C05453=1098.918,347.540,412.649,179.010,19.084,152.317
C05454=1098.913,347.292,412.684,179.007,19.081,152.317
C05455=1098.907,347.044,412.717,179.003,19.078,152.317
C05456=1098.902,346.797,412.751,179.000,19.074,152.316
C05457=1098.895,346.549,412.786,178.998,19.071,152.316
C05458=1098.890,346.301,412.819,178.994,19.067,152.316
C05459=1098.884,346.054,412.853,178.992,19.064,152.316
C05460=1098.879,345.806,412.888,178.988,19.060,152.315
C05461=1098.873,345.558,412.921,178.985,19.057,152.315
C05462=1098.867,345.311,412.955,178.982,19.053,152.315
C05463=1098.862,345.063,412.989,178.979,19.050,152.314
C05464=1098.856,344.816,413.023,178.976,19.046,152.314
C05465=1098.850,344.568,413.056,178.973,19.043,152.314
C05466=1098.844,344.320,413.090,178.969,19.039,152.314
C05467=1098.839,344.073,413.123,178.966,19.036,152.313
C05468=1098.829,343.698,413.175,178.962,19.031,152.313
C05469=1098.821,343.324,413.226,178.957,19.026,152.313
C05470=1098.812,342.950,413.276,178.952,19.021,152.312
C05471=1098.804,342.576,413.327,178.947,19.015,152.312
C05472=1098.798,342.328,413.360,178.945,19.012,152.312
C05473=1098.793,342.080,413.394,178.941,19.008,152.311
C05474=1098.787,341.833,413.428,178.938,19.006,152.311
C05475=1098.781,341.585,413.461,178.935,19.003,152.311
C05476=1098.776,341.337,413.495,178.932,18.999,152.311
C05477=1098.770,341.089,413.528,178.929,18.996,152.311
C05478=1098.764,340.842,413.562,178.925,18.992,152.310
C05479=1098.759,340.594,413.596,178.923,18.989,152.310
C05480=1098.753,340.346,413.629,178.920,18.986,152.310
C05481=1098.747,340.099,413.662,178.916,18.982,152.310
C05482=1098.741,339.851,413.695,178.913,18.979,152.310
C05483=1098.736,339.603,413.729,178.910,18.975,152.309
C05484=1098.730,339.356,413.763,178.907,18.972,152.309
C05485=1098.724,339.108,413.796,178.904,18.970,152.309
C05486=1098.719,338.860,413.829,178.901,18.966,152.309
C05487=1098.713,338.612,413.863,178.898,18.963,152.308
C05488=1098.707,338.364,413.895,178.895,18.960,152.308
C05489=1098.701,338.116,413.929,178.891,18.956,152.308
C05490=1098.696,337.869,413.962,178.888,18.953,152.308
C05491=1098.690,337.621,413.996,178.885,18.950,152.308
C05492=1098.684,337.374,414.029,178.882,18.947,152.308
C05493=1098.678,337.126,414.062,178.879,18.944,152.307
C05494=1098.672,336.878,414.096,178.875,18.940,152.307
C05495=1098.667,336.630,414.129,178.872,18.937,152.307
C05496=1098.661,336.382,414.162,178.870,18.934,152.307
C05497=1098.656,336.135,414.195,178.866,18.931,152.307
C05498=1098.650,335.887,414.228,178.863,18.928,152.306
C05499=1098.644,335.640,414.261,178.860,18.925,152.306
C05500=1098.638,335.392,414.294,178.856,18.921,152.306
C05501=1098.633,335.144,414.327,178.853,18.919,152.306
C05502=1098.627,334.896,414.359,178.851,18.915,152.306
C05503=1098.621,334.648,414.393,178.848,18.913,152.306
C05504=1098.616,334.400,414.426,178.844,18.909,152.305
C05505=1098.610,334.153,414.458,178.841,18.906,152.305
C05506=1098.604,333.905,414.492,178.838,18.903,152.305
C05507=1098.599,333.657,414.525,178.834,18.900,152.305
C05508=1098.593,333.410,414.558,178.831,18.897,152.305
C05509=1098.587,333.161,414.590,178.829,18.894,152.305
C05510=1098.582,332.913,414.624,178.825,18.891,152.305
C05511=1098.576,332.666,414.656,178.822,18.888,152.304
C05512=1098.570,332.418,414.689,178.819,18.885,152.304
C05513=1098.564,332.170,414.722,178.815,18.881,152.304
C05514=1098.559,331.922,414.755,178.812,18.879,152.304
C05515=1098.553,331.675,414.788,178.809,18.876,152.304
C05516=1098.547,331.427,414.821,178.806,18.873,152.304
C05517=1098.542,331.179,414.853,178.803,18.870,152.304
C05518=1098.535,330.932,414.885,178.800,18.867,152.304
C05519=1098.530,330.684,414.919,178.797,18.864,152.303
C05520=1098.520,330.303,414.969,178.791,18.859,152.303
C05521=1098.511,329.923,415.019,178.787,18.855,152.303
C05522=1098.504,329.542,415.068,178.781,18.851,152.303
C05523=1098.494,329.162,415.119,178.777,18.846,152.303
C05524=1098.488,328.915,415.151,178.774,18.844,152.303
C05525=1098.483,328.666,415.184,178.770,18.840,152.303
C05526=1098.477,328.419,415.216,178.767,18.838,152.303
C05527=1098.471,328.170,415.248,178.764,18.835,152.303
C05528=1098.465,327.923,415.281,178.761,18.832,152.302
C05529=1098.460,327.675,415.313,178.757,18.829,152.302
C05530=1098.454,327.427,415.346,178.754,18.826,152.302
C05531=1098.448,327.179,415.378,178.751,18.823,152.302
C05532=1098.442,326.931,415.411,178.748,18.821,152.302
C05533=1098.437,326.684,415.443,178.745,18.818,152.302
C05534=1098.430,326.436,415.476,178.742,18.815,152.302
C05535=1098.424,326.188,415.508,178.738,18.812,152.302
C05536=1098.420,325.940,415.540,178.735,18.810,152.302
C05537=1098.413,325.693,415.573,178.732,18.807,152.302
C05538=1098.407,325.444,415.605,178.729,18.803,152.302
C05539=1098.402,325.197,415.637,178.726,18.801,152.302
C05540=1098.397,324.949,415.670,178.723,18.798,152.301
C05541=1098.391,324.701,415.702,178.720,18.795,152.301
C05542=1098.385,324.453,415.734,178.717,18.793,152.301
C05543=1098.379,324.206,415.766,178.713,18.790,152.301
C05544=1098.374,323.957,415.799,178.710,18.787,152.301
C05545=1098.368,323.710,415.831,178.707,18.784,152.301
C05546=1098.362,323.461,415.863,178.704,18.781,152.301
C05547=1098.356,323.214,415.895,178.701,18.779,152.301
C05548=1098.351,322.966,415.927,178.698,18.776,152.301
C05549=1098.345,322.718,415.960,178.693,18.773,152.301
C05550=1098.340,322.470,415.991,178.690,18.770,152.301
C05551=1098.334,322.222,416.023,178.687,18.768,152.301
C05552=1098.329,322.012,416.050,178.684,18.765,152.301
C05553=1098.324,321.802,416.078,178.682,18.763,152.301
C05554=1098.320,321.592,416.105,178.679,18.760,152.301
C05555=1098.315,321.381,416.132,178.677,18.759,152.301
C05556=1098.310,321.171,416.159,178.674,18.756,152.301
C05557=1098.306,320.961,416.186,178.671,18.754,152.300
C05558=1098.301,320.751,416.213,178.668,18.752,152.301
C05559=1098.296,320.541,416.240,178.666,18.749,152.300
C05560=1098.290,320.293,416.272,178.663,18.747,152.300
C05561=1098.285,320.045,416.304,178.659,18.744,152.300
C05562=1098.279,319.797,416.336,178.656,18.741,152.300
C05563=1098.273,319.549,416.368,178.653,18.738,152.300
C05564=1098.267,319.301,416.400,178.650,18.736,152.300
C05565=1098.262,319.054,416.432,178.647,18.733,152.300
C05566=1098.256,318.805,416.464,178.644,18.731,152.300
C05567=1098.251,318.558,416.495,178.640,18.728,152.300
C05568=1098.245,318.310,416.527,178.637,18.725,152.300
C05569=1098.239,318.062,416.559,178.634,18.722,152.300
C05570=1098.234,317.814,416.592,178.630,18.720,152.300
C05571=1098.229,317.566,416.623,178.627,18.717,152.300
C05572=1098.223,317.334,416.652,178.624,18.715,152.300
C05573=1098.218,317.104,416.682,178.621,18.712,152.300
C05574=1098.213,316.872,416.712,178.618,18.709,152.300
C05575=1098.207,316.640,416.741,178.616,18.708,152.300
C05576=1098.203,316.409,416.771,178.613,18.705,152.300
C05577=1098.198,316.177,416.800,178.609,18.703,152.300
C05578=1098.191,315.946,416.830,178.606,18.700,152.300
C05579=1098.187,315.715,416.859,178.603,18.698,152.300
C05580=1098.181,315.467,416.891,178.600,18.695,152.300
C05581=1098.176,315.219,416.923,178.597,18.692,152.300
C05582=1098.170,314.971,416.955,178.594,18.690,152.300
C05583=1098.164,314.723,416.986,178.591,18.687,152.300
C05584=1098.158,314.475,417.017,178.587,18.685,152.300
C05585=1098.152,314.227,417.049,178.584,18.682,152.300
C05586=1098.147,313.979,417.080,178.581,18.680,152.300
C05587=1098.141,313.731,417.111,178.578,18.678,152.300
C05588=1098.135,313.484,417.143,178.574,18.675,152.300
C05589=1098.129,313.235,417.174,178.571,18.673,152.300
C05590=1098.123,312.988,417.205,178.568,18.670,152.300
C05591=1098.117,312.740,417.237,178.564,18.668,152.300
C05592=1098.112,312.492,417.268,178.561,18.665,152.300
C05593=1098.106,312.244,417.300,178.558,18.663,152.300
C05594=1098.100,311.995,417.331,178.555,18.661,152.300
C05595=1098.095,311.748,417.362,178.552,18.658,152.300
C05596=1098.089,311.499,417.393,178.548,18.656,152.300
C05597=1098.083,311.252,417.425,178.545,18.653,152.300
C05598=1098.077,311.004,417.456,178.542,18.651,152.300
C05599=1098.072,310.756,417.487,178.539,18.649,152.300
C05600=1098.066,310.508,417.519,178.535,18.646,152.300
C05601=1098.060,310.260,417.549,178.532,18.644,152.300
C05602=1098.055,310.012,417.580,178.528,18.641,152.300
C05603=1098.048,309.765,417.611,178.525,18.639,152.300
C05604=1098.043,309.516,417.643,178.522,18.636,152.300
C05605=1098.037,309.268,417.674,178.519,18.634,152.301
C05606=1098.032,309.020,417.705,178.515,18.632,152.301
C05607=1098.026,308.773,417.736,178.512,18.629,152.301
C05608=1098.020,308.524,417.767,178.509,18.627,152.301
C05609=1098.015,308.276,417.798,178.506,18.624,152.301
C05610=1098.009,308.029,417.829,178.503,18.622,152.301
C05611=1098.003,307.780,417.860,178.499,18.620,152.301
C05612=1097.997,307.532,417.891,178.496,18.617,152.301
C05613=1097.992,307.285,417.922,178.493,18.615,152.301
C05614=1097.986,307.037,417.953,178.490,18.613,152.301
C05615=1097.980,306.788,417.984,178.486,18.610,152.301
C05616=1097.974,306.540,418.014,178.483,18.608,152.301
C05617=1097.969,306.293,418.046,178.480,18.606,152.301
C05618=1097.963,306.045,418.076,178.477,18.604,152.301
C05619=1097.958,305.797,418.107,178.473,18.601,152.301
C05620=1097.952,305.548,418.138,178.470,18.599,152.301
C05621=1097.946,305.301,418.170,178.467,18.597,152.301
C05622=1097.941,305.053,418.200,178.464,18.594,152.301
C05623=1097.935,304.805,418.231,178.460,18.592,152.302
C05624=1097.930,304.557,418.261,178.457,18.590,152.302
C05625=1097.924,304.308,418.293,178.453,18.587,152.302
C05626=1097.918,304.060,418.323,178.450,18.585,152.302
C05627=1097.912,303.813,418.353,178.447,18.582,152.302
C05628=1097.904,303.428,418.402,178.442,18.579,152.302
C05629=1097.895,303.043,418.449,178.437,18.575,152.302
C05630=1097.887,302.658,418.497,178.432,18.572,152.302
C05631=1097.878,302.274,418.545,178.427,18.568,152.302
C05632=1097.872,302.026,418.575,178.424,18.566,152.302
C05633=1097.867,301.778,418.606,178.421,18.564,152.302
C05634=1097.861,301.530,418.636,178.417,18.562,152.302
C05635=1097.855,301.282,418.666,178.414,18.559,152.302
C05636=1097.850,301.034,418.697,178.411,18.557,152.303
C05637=1097.845,300.786,418.727,178.408,18.555,152.303
C05638=1097.839,300.538,418.758,178.404,18.552,152.303
C05639=1097.834,300.290,418.789,178.401,18.550,152.303
C05640=1097.827,300.041,418.819,178.398,18.548,152.303
C05641=1097.821,299.793,418.850,178.395,18.545,152.303
C05642=1097.816,299.545,418.881,178.391,18.543,152.303
C05643=1097.811,299.298,418.911,178.388,18.541,152.303
C05644=1097.805,299.049,418.941,178.385,18.539,152.303
C05645=1097.800,298.801,418.972,178.381,18.537,152.303
C05646=1097.794,298.553,419.002,178.378,18.534,152.303
C05647=1097.788,298.305,419.032,178.375,18.532,152.303
C05648=1097.782,298.057,419.063,178.372,18.530,152.303
C05649=1097.778,297.809,419.093,178.368,18.527,152.304
C05650=1097.772,297.561,419.123,178.365,18.526,152.304
C05651=1097.766,297.313,419.154,178.362,18.523,152.304
C05652=1097.761,297.065,419.183,178.358,18.521,152.304
C05653=1097.755,296.817,419.213,178.355,18.519,152.304
C05654=1097.749,296.569,419.244,178.352,18.517,152.304
C05655=1097.743,296.321,419.274,178.348,18.515,152.304
C05656=1097.738,296.073,419.304,178.345,18.512,152.304
C05657=1097.732,295.825,419.334,178.342,18.510,152.305
C05658=1097.727,295.576,419.364,178.338,18.508,152.305
C05659=1097.721,295.328,419.395,178.335,18.506,152.305
C05660=1097.715,295.081,419.425,178.332,18.504,152.305
C05661=1097.710,294.832,419.455,178.328,18.502,152.305
C05662=1097.704,294.584,419.485,178.325,18.499,152.305
C05663=1097.699,294.336,419.515,178.322,18.498,152.305
C05664=1097.693,294.088,419.545,178.319,18.496,152.305
C05665=1097.687,293.840,419.575,178.316,18.494,152.306
C05666=1097.681,293.592,419.605,178.312,18.492,152.306
C05667=1097.676,293.344,419.635,178.309,18.489,152.306
C05668=1097.670,293.095,419.665,178.306,18.487,152.306
C05669=1097.665,292.847,419.695,178.302,18.485,152.306
C05670=1097.659,292.599,419.725,178.299,18.483,152.306
C05671=1097.652,292.351,419.754,178.296,18.481,152.306
C05672=1097.647,292.103,419.784,178.292,18.479,152.306
C05673=1097.641,291.855,419.814,178.289,18.477,152.307
C05674=1097.635,291.607,419.844,178.286,18.474,152.307
C05675=1097.630,291.359,419.874,178.283,18.473,152.307
C05676=1097.625,291.111,419.903,178.280,18.471,152.307
C05677=1097.619,290.863,419.934,178.276,18.469,152.307
C05678=1097.614,290.615,419.963,178.273,18.467,152.307
C05679=1097.608,290.366,419.993,178.269,18.465,152.307
C05680=1097.600,289.996,420.037,178.264,18.461,152.308
C05681=1097.590,289.625,420.082,178.259,18.458,152.308
C05682=1097.582,289.254,420.126,178.255,18.456,152.308
C05683=1097.574,288.883,420.171,178.250,18.453,152.308
C05684=1097.568,288.635,420.200,178.247,18.451,152.308
C05685=1097.562,288.386,420.229,178.243,18.449,152.309
C05686=1097.557,288.139,420.260,178.240,18.447,152.309
C05687=1097.551,287.890,420.289,178.236,18.445,152.309
C05688=1097.545,287.642,420.318,178.233,18.443,152.309
C05689=1097.539,287.394,420.348,178.230,18.441,152.309
C05690=1097.534,287.145,420.378,178.227,18.439,152.309
C05691=1097.528,286.898,420.406,178.224,18.437,152.310
C05692=1097.522,286.650,420.437,178.220,18.435,152.310
C05693=1097.517,286.402,420.466,178.217,18.433,152.310
C05694=1097.511,286.153,420.496,178.213,18.431,152.310
C05695=1097.505,285.905,420.525,178.210,18.429,152.310
C05696=1097.500,285.657,420.555,178.207,18.427,152.310
C05697=1097.495,285.409,420.584,178.204,18.425,152.311
C05698=1097.488,285.161,420.613,178.200,18.424,152.311
C05699=1097.483,284.912,420.643,178.197,18.421,152.311
C05700=1097.477,284.664,420.672,178.194,18.419,152.311
C05701=1097.471,284.416,420.701,178.190,18.418,152.311
C05702=1097.466,284.168,420.731,178.187,18.415,152.311
C05703=1097.461,283.919,420.760,178.183,18.413,152.312
C05704=1097.455,283.671,420.789,178.181,18.412,152.312
C05705=1097.449,283.423,420.819,178.177,18.410,152.312
C05706=1097.443,283.175,420.848,178.174,18.408,152.312
C05707=1097.438,282.927,420.877,178.171,18.406,152.312
C05708=1097.432,282.679,420.907,178.167,18.404,152.312
C05709=1097.426,282.430,420.935,178.164,18.402,152.313
C05710=1097.422,282.182,420.964,178.161,18.400,152.313
C05711=1097.415,281.934,420.993,178.158,18.398,152.313
C05712=1097.410,281.685,421.023,178.154,18.397,152.313
C05713=1097.405,281.438,421.052,178.151,18.394,152.313
C05714=1097.399,281.190,421.081,178.147,18.392,152.313
C05715=1097.393,280.941,421.110,178.144,18.391,152.314
C05716=1097.387,280.692,421.139,178.142,18.389,152.314
C05717=1097.382,280.445,421.169,178.138,18.387,152.314
C05718=1097.376,280.197,421.198,178.134,18.385,152.314
C05719=1097.370,279.948,421.226,178.131,18.383,152.314
C05720=1097.365,279.699,421.256,178.127,18.381,152.315
C05721=1097.359,279.452,421.284,178.125,18.380,152.315
C05722=1097.353,279.203,421.314,178.122,18.378,152.315
C05723=1097.347,278.955,421.342,178.118,18.376,152.315
C05724=1097.343,278.707,421.372,178.115,18.374,152.315
C05725=1097.336,278.459,421.401,178.111,18.372,152.316
C05726=1097.330,278.210,421.429,178.109,18.371,152.316
C05727=1097.325,277.962,421.458,178.105,18.369,152.316
C05728=1097.319,277.714,421.487,178.102,18.367,152.316
C05729=1097.314,277.465,421.516,178.098,18.365,152.316
C05730=1097.308,277.218,421.545,178.095,18.363,152.316
C05731=1097.302,276.969,421.573,178.092,18.361,152.317
C05732=1097.294,276.607,421.615,178.087,18.359,152.317
C05733=1097.286,276.247,421.657,178.082,18.356,152.317
C05734=1097.278,275.884,421.699,178.077,18.353,152.318
C05735=1097.270,275.523,421.741,178.072,18.350,152.318
C05736=1097.264,275.274,421.770,178.069,18.349,152.318
C05737=1097.258,275.026,421.799,178.066,18.347,152.318
C05738=1097.253,274.778,421.827,178.062,18.345,152.319
C05739=1097.247,274.530,421.856,178.059,18.344,152.319
C05740=1097.242,274.282,421.884,178.056,18.342,152.319
C05741=1097.236,274.034,421.913,178.053,18.340,152.319
C05742=1097.230,273.786,421.941,178.049,18.338,152.319
C05743=1097.224,273.537,421.970,178.046,18.336,152.320
C05744=1097.219,273.288,421.999,178.042,18.334,152.320
C05745=1097.214,273.040,422.027,178.040,18.333,152.320
C05746=1097.208,272.792,422.056,178.036,18.331,152.320
C05747=1097.202,272.544,422.084,178.033,18.330,152.321
C05748=1097.196,272.295,422.113,178.029,18.328,152.321
C05749=1097.190,272.047,422.141,178.026,18.326,152.321
C05750=1097.185,271.799,422.170,178.023,18.325,152.321
C05751=1097.179,271.550,422.199,178.019,18.323,152.321
C05752=1097.174,271.302,422.226,178.016,18.321,152.322
C05753=1097.168,271.053,422.255,178.014,18.319,152.322
C05754=1097.162,270.806,422.283,178.010,18.317,152.322
C05755=1097.156,270.557,422.312,178.006,18.315,152.322
C05756=1097.151,270.309,422.340,178.003,18.314,152.322
C05757=1097.145,270.060,422.368,178.000,18.312,152.323
C05758=1097.140,269.813,422.397,177.997,18.310,152.323
C05759=1097.134,269.564,422.426,177.993,18.309,152.323
C05760=1097.129,269.316,422.454,177.990,18.307,152.323
C05761=1097.123,269.067,422.482,177.987,18.305,152.324
C05762=1097.118,268.819,422.510,177.984,18.304,152.324
C05763=1097.112,268.570,422.538,177.980,18.302,152.324
C05764=1097.106,268.322,422.566,177.977,18.300,152.324
C05765=1097.100,268.073,422.595,177.974,18.299,152.324
C05766=1097.095,267.825,422.622,177.970,18.297,152.325
C05767=1097.089,267.577,422.652,177.967,18.295,152.325
C05768=1097.083,267.329,422.679,177.964,18.294,152.325
C05769=1097.078,267.080,422.708,177.961,18.292,152.325
C05770=1097.072,266.832,422.736,177.957,18.290,152.326
C05771=1097.066,266.584,422.764,177.953,18.289,152.326
C05772=1097.061,266.336,422.792,177.951,18.287,152.326
C05773=1097.056,266.088,422.820,177.947,18.285,152.326
C05774=1097.050,265.839,422.848,177.944,18.284,152.327
C05775=1097.044,265.591,422.876,177.940,18.282,152.327
C05776=1097.038,265.342,422.903,177.937,18.280,152.327
C05777=1097.033,265.094,422.931,177.934,18.279,152.327
C05778=1097.027,264.845,422.960,177.930,18.277,152.328
C05779=1097.021,264.597,422.988,177.928,18.276,152.328
C05780=1097.016,264.349,423.015,177.924,18.274,152.328
C05781=1097.010,264.100,423.044,177.921,18.272,152.328
C05782=1097.005,263.852,423.072,177.917,18.270,152.329
C05783=1096.998,263.604,423.100,177.914,18.269,152.329
C05784=1096.990,263.245,423.140,177.909,18.266,152.329
C05785=1096.981,262.886,423.180,177.904,18.264,152.330
C05786=1096.973,262.527,423.220,177.900,18.262,152.330
C05787=1096.965,262.168,423.260,177.895,18.259,152.330
C05788=1096.960,261.920,423.287,177.892,18.258,152.331
C05789=1096.954,261.671,423.316,177.888,18.257,152.331
C05790=1096.948,261.424,423.343,177.885,18.255,152.331
C05791=1096.942,261.174,423.371,177.882,18.253,152.331
C05792=1096.937,260.926,423.399,177.879,18.252,152.332
C05793=1096.931,260.679,423.426,177.875,18.250,152.332
C05794=1096.925,260.429,423.454,177.872,18.249,152.332
C05795=1096.920,260.181,423.482,177.869,18.247,152.333
C05796=1096.913,259.933,423.509,177.865,18.245,152.333
C05797=1096.908,259.684,423.537,177.862,18.244,152.333
C05798=1096.903,259.436,423.565,177.859,18.243,152.333
C05799=1096.897,259.188,423.591,177.855,18.241,152.334
C05800=1096.891,258.939,423.620,177.852,18.239,152.334
C05801=1096.885,258.691,423.648,177.849,18.238,152.334
C05802=1096.880,258.442,423.674,177.845,18.236,152.334
C05803=1096.874,258.194,423.703,177.842,18.235,152.335
C05804=1096.868,257.945,423.729,177.839,18.233,152.335
C05805=1096.863,257.697,423.757,177.835,18.231,152.335
C05806=1096.857,257.448,423.785,177.833,18.230,152.335
C05807=1096.851,257.200,423.812,177.829,18.229,152.336
C05808=1096.846,256.951,423.839,177.825,18.227,152.336
C05809=1096.840,256.704,423.867,177.823,18.226,152.336
C05810=1096.834,256.454,423.894,177.819,18.224,152.336
C05811=1096.829,256.206,423.922,177.816,18.222,152.337
C05812=1096.823,255.958,423.949,177.813,18.221,152.337
C05813=1096.817,255.709,423.977,177.809,18.219,152.337
C05814=1096.811,255.461,424.004,177.806,18.217,152.338
C05815=1096.806,255.212,424.031,177.803,18.216,152.338
C05816=1096.800,254.964,424.058,177.799,18.215,152.338
C05817=1096.795,254.716,424.086,177.796,18.213,152.338
C05818=1096.789,254.467,424.113,177.793,18.212,152.339
C05819=1096.783,254.219,424.141,177.789,18.210,152.339
C05820=1096.778,253.970,424.167,177.787,18.208,152.339
C05821=1096.773,253.722,424.195,177.783,18.207,152.340
C05822=1096.767,253.474,424.222,177.779,18.205,152.340
C05823=1096.761,253.224,424.250,177.777,18.204,152.340
C05824=1096.755,252.976,424.276,177.773,18.202,152.340
C05825=1096.750,252.727,424.303,177.770,18.200,152.340
C05826=1096.744,252.480,424.331,177.767,18.199,152.341
C05827=1096.739,252.231,424.358,177.763,18.198,152.341
C05828=1096.733,251.983,424.385,177.760,18.196,152.341
C05829=1096.728,251.733,424.412,177.757,18.195,152.342
C05830=1096.722,251.485,424.439,177.753,18.193,152.342
C05831=1096.716,251.237,424.467,177.751,18.192,152.342
C05832=1096.711,250.989,424.494,177.747,18.190,152.342
C05833=1096.706,250.740,424.521,177.744,18.188,152.343
C05834=1096.700,250.492,424.547,177.741,18.187,152.343
C05835=1096.694,250.243,424.574,177.737,18.186,152.343
C05836=1096.686,249.881,424.614,177.733,18.183,152.344
C05837=1096.679,249.520,424.653,177.727,18.181,152.344
C05838=1096.670,249.158,424.692,177.723,18.179,152.344
C05839=1096.662,248.796,424.732,177.718,18.177,152.345
C05840=1096.656,248.548,424.759,177.715,18.175,152.345
C05841=1096.651,248.299,424.786,177.712,18.174,152.345
C05842=1096.645,248.051,424.813,177.708,18.172,152.346
C05843=1096.640,247.803,424.839,177.706,18.170,152.346
C05844=1096.635,247.554,424.866,177.702,18.169,152.346
C05845=1096.629,247.306,424.893,177.698,18.167,152.346
C05846=1096.623,247.057,424.920,177.696,18.166,152.347
C05847=1096.618,246.808,424.946,177.692,18.165,152.347
C05848=1096.612,246.559,424.973,177.689,18.163,152.347
C05849=1096.607,246.311,425.000,177.686,18.161,152.348
C05850=1096.601,246.063,425.026,177.682,18.160,152.348
C05851=1096.595,245.814,425.053,177.679,18.159,152.348
C05852=1096.590,245.566,425.080,177.676,18.157,152.348
C05853=1096.584,245.317,425.107,177.673,18.156,152.349
C05854=1096.579,245.069,425.133,177.669,18.154,152.349
C05855=1096.573,244.821,425.160,177.666,18.153,152.349
C05856=1096.567,244.572,425.186,177.663,18.151,152.350
C05857=1096.562,244.323,425.213,177.659,18.150,152.350
C05858=1096.557,244.075,425.240,177.657,18.149,152.350
C05859=1096.551,243.826,425.267,177.653,18.147,152.350
C05860=1096.545,243.577,425.293,177.650,18.146,152.351
C05861=1096.540,243.329,425.319,177.647,18.144,152.351
C05862=1096.534,243.081,425.346,177.643,18.142,152.351
C05863=1096.528,242.832,425.372,177.640,18.141,152.352
C05864=1096.523,242.583,425.398,177.637,18.140,152.352
C05865=1096.517,242.335,425.425,177.634,18.139,152.352
C05866=1096.511,242.087,425.452,177.630,18.137,152.353
C05867=1096.505,241.838,425.478,177.627,18.136,152.353
C05868=1096.500,241.589,425.504,177.624,18.134,152.353
C05869=1096.494,241.341,425.531,177.620,18.133,152.353
C05870=1096.488,241.092,425.557,177.617,18.132,152.354
C05871=1096.483,240.844,425.583,177.614,18.130,152.354
C05872=1096.477,240.595,425.610,177.611,18.129,152.354
C05873=1096.471,240.346,425.636,177.607,18.127,152.355
C05874=1096.466,240.098,425.663,177.604,18.126,152.355
C05875=1096.460,239.849,425.689,177.601,18.125,152.355
C05876=1096.454,239.600,425.715,177.598,18.123,152.356
C05877=1096.449,239.352,425.742,177.594,18.122,152.356
C05878=1096.443,239.103,425.768,177.591,18.120,152.356
C05879=1096.437,238.855,425.795,177.588,18.119,152.356
C05880=1096.432,238.606,425.820,177.584,18.118,152.357
C05881=1096.426,238.357,425.847,177.581,18.116,152.357
C05882=1096.421,238.108,425.873,177.578,18.115,152.357
C05883=1096.415,237.860,425.900,177.575,18.114,152.358
C05884=1096.410,237.612,425.925,177.571,18.112,152.358
C05885=1096.404,237.364,425.951,177.568,18.111,152.358
C05886=1096.398,237.115,425.977,177.565,18.109,152.359
C05887=1096.393,236.866,426.003,177.562,18.108,152.359
C05888=1096.384,236.498,426.042,177.557,18.106,152.359
C05889=1096.376,236.129,426.081,177.552,18.104,152.360
C05890=1096.368,235.760,426.119,177.547,18.102,152.360
C05891=1096.359,235.392,426.158,177.543,18.100,152.361
C05892=1096.354,235.143,426.184,177.539,18.098,152.361
C05893=1096.349,234.895,426.210,177.536,18.097,152.361
C05894=1096.343,234.646,426.236,177.533,18.096,152.362
C05895=1096.337,234.397,426.262,177.530,18.095,152.362
C05896=1096.331,234.149,426.288,177.526,18.093,152.362
C05897=1096.326,233.900,426.314,177.524,18.092,152.362
C05898=1096.320,233.651,426.340,177.520,18.090,152.363
C05899=1096.315,233.403,426.366,177.517,18.089,152.363
C05900=1096.309,233.155,426.392,177.513,18.088,152.363
C05901=1096.303,232.906,426.418,177.511,18.086,152.364
C05902=1096.298,232.657,426.444,177.507,18.085,152.364
C05903=1096.292,232.408,426.469,177.504,18.084,152.364
C05904=1096.287,232.160,426.494,177.500,18.082,152.365
C05905=1096.281,231.911,426.521,177.498,18.081,152.365
C05906=1096.276,231.662,426.547,177.494,18.079,152.365
C05907=1096.269,231.414,426.572,177.491,18.078,152.366
C05908=1096.265,231.165,426.598,177.488,18.077,152.366
C05909=1096.259,230.916,426.624,177.485,18.076,152.366
C05910=1096.253,230.668,426.649,177.481,18.074,152.367
C05911=1096.247,230.419,426.675,177.478,18.073,152.367
C05912=1096.243,230.171,426.701,177.475,18.071,152.367
C05913=1096.236,229.922,426.726,177.472,18.071,152.368
C05914=1096.231,229.674,426.753,177.468,18.069,152.368
C05915=1096.224,229.425,426.778,177.465,18.068,152.368
C05916=1096.220,229.177,426.804,177.462,18.066,152.368
C05917=1096.213,228.928,426.829,177.459,18.065,152.369
C05918=1096.208,228.679,426.855,177.455,18.064,152.369
C05919=1096.202,228.430,426.880,177.452,18.063,152.369
C05920=1096.197,228.182,426.906,177.449,18.061,152.370
C05921=1096.191,227.933,426.931,177.446,18.060,152.370
C05922=1096.185,227.684,426.957,177.442,18.058,152.370
C05923=1096.179,227.435,426.982,177.439,18.057,152.371
C05924=1096.174,227.187,427.007,177.437,18.056,152.371
C05925=1096.168,226.938,427.033,177.433,18.055,152.371
C05926=1096.163,226.689,427.058,177.430,18.054,152.372
C05927=1096.157,226.441,427.083,177.426,18.052,152.372
C05928=1096.152,226.192,427.109,177.424,18.051,152.372
C05929=1096.145,225.943,427.135,177.420,18.050,152.373
C05930=1096.141,225.695,427.160,177.417,18.048,152.373
C05931=1096.134,225.447,427.186,177.413,18.047,152.373
C05932=1096.129,225.197,427.211,177.411,18.046,152.374
C05933=1096.124,224.949,427.236,177.407,18.044,152.374
C05934=1096.118,224.700,427.262,177.404,18.043,152.374
C05935=1096.113,224.452,427.287,177.400,18.042,152.375
C05936=1096.106,224.203,427.312,177.398,18.041,152.375
C05937=1096.101,223.954,427.337,177.395,18.040,152.375
C05938=1096.096,223.706,427.362,177.391,18.038,152.376
C05939=1096.090,223.457,427.388,177.388,18.037,152.376
C05940=1096.082,223.080,427.426,177.383,18.035,152.376
C05941=1096.073,222.702,427.464,177.378,18.033,152.377
C05942=1096.064,222.326,427.502,177.373,18.031,152.377
C05943=1096.056,221.948,427.541,177.369,18.029,152.378
C05944=1096.051,221.700,427.566,177.365,18.027,152.378
C05945=1096.045,221.451,427.590,177.362,18.027,152.378
C05946=1096.039,221.202,427.616,177.359,18.026,152.379
C05947=1096.034,220.954,427.641,177.356,18.024,152.379
C05948=1096.028,220.705,427.666,177.353,18.023,152.380
C05949=1096.022,220.457,427.691,177.349,18.021,152.380
C05950=1096.017,220.207,427.716,177.346,18.021,152.380
C05951=1096.011,219.959,427.741,177.343,18.019,152.380
C05952=1096.005,219.710,427.766,177.340,18.018,152.381
C05953=1095.999,219.461,427.791,177.337,18.017,152.381
C05954=1095.994,219.213,427.817,177.333,18.015,152.381
C05955=1095.988,218.964,427.841,177.330,18.015,152.382
C05956=1095.983,218.716,427.866,177.327,18.013,152.382
C05957=1095.977,218.466,427.891,177.324,18.012,152.383
C05958=1095.971,218.218,427.916,177.321,18.011,152.383
C05959=1095.965,217.969,427.940,177.317,18.009,152.383
C05960=1095.961,217.720,427.965,177.315,18.008,152.383
C05961=1095.955,217.472,427.991,177.311,18.007,152.384
C05962=1095.949,217.223,428.015,177.308,18.006,152.384
C05963=1095.943,216.974,428.040,177.305,18.005,152.384
C05964=1095.938,216.726,428.064,177.301,18.003,152.385
C05965=1095.932,216.477,428.090,177.299,18.002,152.385
C05966=1095.927,216.228,428.115,177.295,18.001,152.386
C05967=1095.921,215.979,428.139,177.292,18.000,152.386
C05968=1095.916,215.731,428.164,177.289,17.999,152.386
C05969=1095.910,215.482,428.189,177.286,17.997,152.386
C05970=1095.904,215.233,428.213,177.283,17.996,152.387
C05971=1095.899,214.985,428.238,177.279,17.994,152.387
C05972=1095.893,214.736,428.263,177.276,17.994,152.387
C05973=1095.888,214.487,428.287,177.274,17.992,152.388
C05974=1095.881,214.239,428.312,177.270,17.991,152.388
C05975=1095.877,213.990,428.337,177.267,17.990,152.388
C05976=1095.871,213.740,428.362,177.263,17.988,152.389
C05977=1095.866,213.492,428.386,177.260,17.988,152.389
C05978=1095.860,213.244,428.411,177.258,17.986,152.389
C05979=1095.854,212.995,428.436,177.254,17.985,152.390
C05980=1095.849,212.746,428.460,177.251,17.984,152.390
C05981=1095.843,212.497,428.484,177.248,17.983,152.390
C05982=1095.838,212.248,428.509,177.245,17.981,152.391
C05983=1095.832,212.000,428.534,177.242,17.980,152.391
C05984=1095.826,211.751,428.558,177.238,17.979,152.392
C05985=1095.821,211.502,428.583,177.235,17.978,152.392
C05986=1095.814,211.253,428.607,177.232,17.977,152.392
C05987=1095.809,211.005,428.631,177.229,17.975,152.392
C05988=1095.804,210.756,428.655,177.226,17.974,152.393
C05989=1095.798,210.507,428.680,177.223,17.973,152.393
C05990=1095.792,210.258,428.704,177.219,17.972,152.393
C05991=1095.787,210.010,428.729,177.216,17.971,152.394
C05992=1095.778,209.636,428.765,177.212,17.969,152.394
C05993=1095.770,209.263,428.802,177.207,17.967,152.395
C05994=1095.761,208.890,428.838,177.202,17.966,152.395
C05995=1095.753,208.516,428.874,177.198,17.964,152.396
C05996=1095.730,207.502,428.973,177.146,17.942,152.401
C05997=1095.724,207.253,428.997,177.143,17.942,152.402
C05998=1095.718,207.005,429.021,177.139,17.942,152.402
C05999=1095.713,206.756,429.045,177.136,17.942,152.403
C06000=1095.708,206.507,429.069,177.133,17.941,152.403
C06001=1095.702,206.259,429.092,177.129,17.940,152.404
C06002=1095.696,206.010,429.117,177.126,17.940,152.404
C06003=1095.690,205.761,429.141,177.122,17.940,152.405
C06004=1095.685,205.512,429.164,177.119,17.939,152.405
C06005=1095.680,205.263,429.188,177.116,17.939,152.406
C06006=1095.674,205.015,429.212,177.113,17.939,152.406
C06007=1095.668,204.765,429.236,177.109,17.938,152.407
C06008=1095.663,204.517,429.260,177.106,17.938,152.408
C06009=1095.657,204.268,429.284,177.103,17.938,152.408
C06010=1095.652,204.019,429.307,177.100,17.938,152.409
C06011=1095.646,203.771,429.331,177.096,17.937,152.409
C06012=1095.641,203.522,429.355,177.093,17.937,152.410
C06013=1095.635,203.272,429.379,177.090,17.937,152.410
C06014=1095.629,203.024,429.403,177.087,17.936,152.411
C06015=1095.624,202.776,429.427,177.083,17.936,152.411
C06016=1095.618,202.527,429.450,177.080,17.936,152.412
C06017=1095.613,202.278,429.474,177.077,17.936,152.413
C06018=1095.607,202.029,429.497,177.073,17.936,152.413
C06019=1095.600,201.780,429.521,177.070,17.935,152.414
C06020=1095.595,201.531,429.545,177.067,17.935,152.414
C06021=1095.589,201.283,429.569,177.064,17.935,152.415
C06022=1095.584,201.033,429.592,177.060,17.934,152.415
C06023=1095.578,200.785,429.616,177.057,17.934,152.416
C06024=1095.572,200.536,429.639,177.053,17.933,152.416
C06025=1095.567,200.287,429.663,177.050,17.933,152.417
C06026=1095.561,200.038,429.686,177.047,17.932,152.418
C06027=1095.555,199.790,429.710,177.043,17.932,152.418
C06028=1095.550,199.541,429.733,177.040,17.932,152.419
C06029=1095.544,199.292,429.757,177.037,17.932,152.419
C06030=1095.539,199.043,429.781,177.034,17.931,152.420
C06031=1095.533,198.795,429.804,177.030,17.931,152.420
C06032=1095.526,198.545,429.828,177.027,17.931,152.421
C06033=1095.521,198.296,429.851,177.024,17.930,152.421
C06034=1095.515,198.048,429.875,177.021,17.930,152.422
C06035=1095.510,197.799,429.898,177.017,17.930,152.423
C06036=1095.505,197.550,429.921,177.014,17.929,152.423
C06037=1095.499,197.301,429.945,177.011,17.929,152.424
C06038=1095.493,197.053,429.968,177.008,17.929,152.424
C06039=1095.488,196.803,429.991,177.004,17.929,152.425
C06040=1095.482,196.555,430.015,177.001,17.928,152.425
C06041=1095.476,196.306,430.038,176.998,17.928,152.426
C06042=1095.470,196.057,430.061,176.995,17.928,152.426
C06043=1095.465,195.809,430.085,176.991,17.927,152.427
C06044=1095.459,195.560,430.108,176.988,17.927,152.427
C06045=1095.454,195.311,430.131,176.985,17.927,152.428
C06046=1095.449,195.062,430.155,176.982,17.926,152.429
C06047=1095.443,194.813,430.178,176.978,17.926,152.429
C06048=1095.436,194.564,430.202,176.975,17.925,152.430
C06049=1095.431,194.315,430.225,176.972,17.925,152.430
C06050=1095.426,194.066,430.248,176.969,17.925,152.431
C06051=1095.420,193.817,430.271,176.966,17.924,152.431
C06052=1095.414,193.569,430.294,176.962,17.924,152.432
C06053=1095.409,193.320,430.317,176.959,17.924,152.432
C06054=1095.404,193.071,430.341,176.956,17.924,152.433
C06055=1095.398,192.822,430.364,176.953,17.923,152.433
C06056=1095.392,192.573,430.387,176.950,17.923,152.434
C06057=1095.385,192.299,430.412,176.946,17.923,152.434
C06058=1095.379,192.023,430.439,176.943,17.922,152.435
C06059=1095.374,191.749,430.463,176.939,17.922,152.436
C06060=1095.368,191.474,430.489,176.936,17.921,152.436
C06061=1095.362,191.225,430.512,176.932,17.921,152.437
C06062=1095.356,190.976,430.535,176.929,17.920,152.437
C06063=1095.350,190.727,430.558,176.926,17.920,152.438
C06064=1095.345,190.478,430.582,176.923,17.920,152.438
C06065=1095.340,190.229,430.605,176.920,17.919,152.439
C06066=1095.334,189.980,430.628,176.916,17.919,152.439
C06067=1095.328,189.731,430.651,176.913,17.918,152.440
C06068=1095.323,189.483,430.673,176.910,17.918,152.440
C06069=1095.317,189.234,430.696,176.907,17.918,152.441
C06070=1095.312,188.985,430.720,176.904,17.917,152.441
C06071=1095.307,188.736,430.743,176.901,17.917,152.442
C06072=1095.301,188.487,430.766,176.897,17.916,152.442
C06073=1095.295,188.238,430.788,176.894,17.916,152.443
C06074=1095.289,187.989,430.811,176.891,17.915,152.443
C06075=1095.284,187.741,430.834,176.888,17.915,152.444
C06076=1095.279,187.492,430.857,176.885,17.915,152.444
C06077=1095.274,187.242,430.880,176.882,17.915,152.445
C06078=1095.268,186.993,430.903,176.879,17.914,152.445
C06079=1095.262,186.745,430.926,176.876,17.914,152.446
C06080=1095.257,186.496,430.949,176.873,17.914,152.446
C06081=1095.252,186.247,430.971,176.870,17.913,152.447
C06082=1095.246,185.999,430.994,176.867,17.913,152.447
C06083=1095.240,185.749,431.016,176.863,17.912,152.448
C06084=1095.235,185.500,431.039,176.860,17.911,152.448
C06085=1095.229,185.251,431.062,176.857,17.911,152.449
C06086=1095.224,185.003,431.085,176.854,17.911,152.449
C06087=1095.218,184.754,431.108,176.851,17.910,152.450
C06088=1095.213,184.505,431.130,176.848,17.910,152.450
C06089=1095.207,184.256,431.153,176.844,17.910,152.451
C06090=1095.200,184.007,431.175,176.841,17.909,152.452
C06091=1095.195,183.758,431.198,176.838,17.909,152.452
C06092=1095.189,183.509,431.220,176.835,17.909,152.453
C06093=1095.184,183.260,431.243,176.832,17.908,152.453
C06094=1095.178,183.011,431.266,176.828,17.908,152.454
C06095=1095.172,182.763,431.288,176.826,17.908,152.454
C06096=1095.167,182.514,431.311,176.823,17.908,152.455
C06097=1095.161,182.265,431.334,176.819,17.907,152.455
C06098=1095.155,182.016,431.356,176.816,17.907,152.456
C06099=1095.149,181.767,431.378,176.813,17.906,152.456
C06100=1095.143,181.518,431.401,176.810,17.906,152.457
C06101=1095.137,181.269,431.424,176.807,17.906,152.457
C06102=1095.133,181.020,431.446,176.804,17.905,152.458
C06103=1095.126,180.771,431.468,176.800,17.905,152.458
C06104=1095.121,180.522,431.490,176.797,17.904,152.459
C06105=1095.115,180.273,431.513,176.794,17.904,152.459
C06106=1095.109,180.024,431.536,176.791,17.903,152.460
C06107=1095.104,179.776,431.558,176.788,17.903,152.460
C06108=1095.098,179.527,431.581,176.784,17.903,152.461
C06109=1095.093,179.277,431.603,176.782,17.903,152.461
C06110=1095.086,179.029,431.625,176.779,17.902,152.462
C06111=1095.081,178.780,431.647,176.776,17.902,152.462
C06112=1095.076,178.531,431.670,176.773,17.901,152.463
C06113=1095.069,178.282,431.692,176.770,17.901,152.463
C06114=1095.064,178.033,431.715,176.766,17.901,152.464
C06115=1095.058,177.783,431.737,176.763,17.900,152.464
C06116=1095.052,177.535,431.759,176.760,17.900,152.465
C06117=1095.047,177.286,431.781,176.757,17.899,152.465
C06118=1095.041,177.037,431.804,176.754,17.899,152.466
C06119=1095.036,176.788,431.825,176.751,17.898,152.466
C06120=1095.030,176.539,431.847,176.748,17.898,152.467
C06121=1095.024,176.264,431.872,176.744,17.897,152.467
C06122=1095.018,175.989,431.897,176.741,17.897,152.468
C06123=1095.011,175.713,431.922,176.738,17.897,152.468
C06124=1095.005,175.438,431.945,176.735,17.897,152.469
C06125=1094.999,175.190,431.968,176.732,17.896,152.469
C06126=1094.994,174.940,431.990,176.728,17.896,152.470
C06127=1094.988,174.691,432.013,176.725,17.895,152.470
C06128=1094.983,174.443,432.034,176.722,17.895,152.471
C06129=1094.977,174.193,432.057,176.719,17.894,152.471
C06130=1094.971,173.944,432.078,176.716,17.894,152.472
C06131=1094.966,173.696,432.101,176.713,17.893,152.472
C06132=1094.960,173.447,432.122,176.710,17.893,152.473
C06133=1094.954,173.197,432.145,176.707,17.892,152.473
C06134=1094.949,172.949,432.167,176.704,17.892,152.474
C06135=1094.943,172.700,432.189,176.701,17.891,152.474
C06136=1094.938,172.450,432.211,176.698,17.891,152.475
C06137=1094.932,172.202,432.232,176.695,17.890,152.475
C06138=1094.926,171.953,432.255,176.692,17.890,152.476
C06139=1094.921,171.704,432.277,176.689,17.889,152.476
C06140=1094.915,171.455,432.299,176.685,17.889,152.477
C06141=1094.909,171.205,432.320,176.683,17.889,152.477
C06142=1094.904,170.957,432.342,176.680,17.889,152.478
C06143=1094.898,170.707,432.364,176.677,17.888,152.478
C06144=1094.893,170.459,432.387,176.674,17.887,152.478
C06145=1094.888,170.210,432.409,176.671,17.887,152.479
C06146=1094.882,169.961,432.430,176.668,17.886,152.479
C06147=1094.877,169.712,432.452,176.665,17.886,152.480
C06148=1094.871,169.463,432.474,176.662,17.885,152.480
C06149=1094.866,169.214,432.496,176.659,17.885,152.481
C06150=1094.860,168.964,432.517,176.656,17.885,152.481
C06151=1094.855,168.716,432.539,176.653,17.884,152.482
C06152=1094.849,168.466,432.561,176.650,17.883,152.482
C06153=1094.843,168.218,432.584,176.647,17.883,152.483
C06154=1094.837,167.969,432.605,176.644,17.882,152.483
C06155=1094.832,167.720,432.627,176.641,17.881,152.483
C06156=1094.826,167.471,432.649,176.638,17.881,152.484
C06157=1094.822,167.222,432.671,176.636,17.881,152.484
C06158=1094.815,166.973,432.692,176.633,17.880,152.485
C06159=1094.810,166.725,432.713,176.629,17.880,152.485
C06160=1094.804,166.475,432.736,176.626,17.879,152.486
C06161=1094.799,166.227,432.757,176.623,17.878,152.486
C06162=1094.793,165.977,432.779,176.620,17.878,152.487
C06163=1094.788,165.728,432.800,176.617,17.877,152.487
C06164=1094.783,165.479,432.822,176.614,17.877,152.488
C06165=1094.777,165.230,432.843,176.612,17.877,152.488
C06166=1094.772,164.981,432.865,176.609,17.876,152.488
C06167=1094.766,164.732,432.887,176.606,17.876,152.489
C06168=1094.761,164.483,432.908,176.603,17.875,152.489
C06169=1094.755,164.234,432.930,176.600,17.874,152.490
C06170=1094.750,163.985,432.951,176.597,17.873,152.490
C06171=1094.745,163.736,432.973,176.593,17.873,152.491
C06172=1094.739,163.487,432.995,176.591,17.873,152.491
C06173=1094.733,163.238,433.016,176.588,17.872,152.492
C06174=1094.728,162.989,433.038,176.585,17.871,152.492
C06175=1094.722,162.740,433.059,176.582,17.871,152.492
C06176=1094.718,162.491,433.081,176.579,17.870,152.493
C06177=1094.711,162.242,433.103,176.576,17.870,152.493
C06178=1094.706,161.993,433.123,176.573,17.869,152.494
C06179=1094.701,161.743,433.145,176.571,17.869,152.494
C06180=1094.695,161.495,433.167,176.568,17.868,152.494
C06181=1094.690,161.246,433.188,176.565,17.867,152.495
C06182=1094.684,160.997,433.209,176.562,17.867,152.495
C06183=1094.679,160.748,433.231,176.559,17.866,152.496
C06184=1094.673,160.499,433.252,176.556,17.866,152.496
C06185=1094.666,160.224,433.275,176.552,17.865,152.497
C06186=1094.660,159.948,433.300,176.549,17.865,152.497
C06187=1094.654,159.673,433.323,176.546,17.864,152.498
C06188=1094.647,159.396,433.346,176.543,17.864,152.498
C06189=1094.643,159.147,433.368,176.540,17.863,152.499
C06190=1094.636,158.898,433.389,176.537,17.862,152.499
C06191=1094.631,158.649,433.410,176.534,17.862,152.500
C06192=1094.625,158.400,433.431,176.532,17.862,152.500
C06193=1094.619,158.151,433.453,176.529,17.861,152.500
C06194=1094.614,157.902,433.473,176.526,17.860,152.501
C06195=1094.608,157.653,433.495,176.523,17.860,152.501
C06196=1094.603,157.404,433.515,176.520,17.859,152.502
C06197=1094.597,157.155,433.537,176.517,17.859,152.502
C06198=1094.592,156.906,433.559,176.514,17.858,152.503
C06199=1094.587,156.657,433.580,176.511,17.858,152.503
C06200=1094.581,156.408,433.601,176.508,17.857,152.503
C06201=1094.575,156.159,433.622,176.505,17.856,152.504
C06202=1094.570,155.910,433.643,176.503,17.855,152.504
C06203=1094.564,155.661,433.664,176.500,17.855,152.505
C06204=1094.558,155.412,433.685,176.497,17.855,152.505
C06205=1094.553,155.163,433.706,176.494,17.854,152.506
C06206=1094.547,154.913,433.727,176.491,17.854,152.506
C06207=1094.542,154.664,433.748,176.488,17.853,152.506
C06208=1094.536,154.416,433.769,176.486,17.853,152.507
C06209=1094.530,154.166,433.790,176.483,17.852,152.507
C06210=1094.525,153.917,433.811,176.480,17.851,152.508
C06211=1094.519,153.668,433.832,176.477,17.850,152.508
C06212=1094.514,153.420,433.853,176.474,17.850,152.508
C06213=1094.508,153.170,433.874,176.472,17.850,152.509
C06214=1094.502,152.921,433.895,176.469,17.849,152.509
C06215=1094.497,152.672,433.916,176.466,17.849,152.510
C06216=1094.490,152.423,433.936,176.463,17.848,152.510
C06217=1094.485,152.174,433.958,176.460,17.847,152.511
C06218=1094.480,151.925,433.978,176.457,17.847,152.511
C06219=1094.473,151.676,434.000,176.454,17.846,152.511
C06220=1094.468,151.427,434.020,176.451,17.846,152.512
C06221=1094.463,151.178,434.041,176.448,17.845,152.512
C06222=1094.457,150.929,434.062,176.445,17.844,152.513
C06223=1094.452,150.679,434.083,176.443,17.844,152.513
C06224=1094.446,150.430,434.104,176.440,17.843,152.513
C06225=1094.441,150.182,434.125,176.437,17.842,152.514
C06226=1094.435,149.933,434.145,176.434,17.842,152.514
C06227=1094.429,149.683,434.166,176.431,17.841,152.515
C06228=1094.424,149.434,434.186,176.429,17.841,152.515
C06229=1094.418,149.186,434.208,176.426,17.840,152.515
C06230=1094.413,148.936,434.228,176.423,17.839,152.516
C06231=1094.408,148.687,434.249,176.420,17.839,152.516
C06232=1094.402,148.437,434.270,176.417,17.838,152.517
C06233=1094.395,148.189,434.290,176.415,17.838,152.517
C06234=1094.390,147.940,434.311,176.412,17.837,152.518
C06235=1094.385,147.691,434.331,176.409,17.836,152.518
C06236=1094.379,147.441,434.352,176.406,17.836,152.518
C06237=1094.373,147.192,434.372,176.404,17.835,152.519
C06238=1094.367,146.944,434.394,176.401,17.834,152.519
C06239=1094.362,146.695,434.414,176.398,17.833,152.519
C06240=1094.356,146.445,434.434,176.395,17.833,152.520
C06241=1094.350,146.196,434.455,176.392,17.832,152.520
C06242=1094.345,145.947,434.475,176.390,17.832,152.521
C06243=1094.340,145.698,434.496,176.387,17.831,152.521
C06244=1094.334,145.449,434.516,176.384,17.830,152.521
C06245=1094.328,145.200,434.538,176.381,17.830,152.522
C06246=1094.322,144.951,434.558,176.379,17.830,152.522
C06247=1094.316,144.702,434.578,176.376,17.829,152.523
C06248=1094.311,144.453,434.599,176.373,17.828,152.523
C06249=1094.305,144.177,434.621,176.370,17.827,152.523
C06250=1094.299,143.901,434.644,176.367,17.827,152.524
C06251=1094.293,143.625,434.667,176.364,17.826,152.524
C06252=1094.287,143.350,434.689,176.361,17.825,152.525
C06253=1094.281,143.100,434.710,176.358,17.825,152.525
C06254=1094.275,142.851,434.730,176.355,17.823,152.525
C06255=1094.270,142.602,434.751,176.353,17.823,152.526
C06256=1094.264,142.353,434.771,176.350,17.822,152.526
C06257=1094.258,142.104,434.791,176.347,17.822,152.527
C06258=1094.253,141.855,434.812,176.344,17.821,152.527
C06259=1094.248,141.606,434.832,176.341,17.820,152.527
C06260=1094.242,141.357,434.852,176.339,17.820,152.528
C06261=1094.237,141.108,434.873,176.336,17.819,152.528
C06262=1094.230,140.858,434.893,176.333,17.818,152.529
C06263=1094.225,140.609,434.914,176.330,17.817,152.529
C06264=1094.220,140.359,434.933,176.328,17.817,152.529
C06265=1094.214,140.111,434.953,176.325,17.816,152.530
C06266=1094.209,139.861,434.974,176.322,17.815,152.530
C06267=1094.203,139.613,434.994,176.319,17.815,152.530
C06268=1094.197,139.363,435.014,176.317,17.814,152.531
C06269=1094.191,139.115,435.034,176.314,17.813,152.531
C06270=1094.186,138.866,435.055,176.311,17.813,152.531
C06271=1094.180,138.617,435.075,176.308,17.812,152.532
C06272=1094.175,138.367,435.095,176.307,17.811,152.532
C06273=1094.168,138.117,435.115,176.304,17.811,152.533
C06274=1094.163,137.868,435.136,176.301,17.810,152.533
C06275=1094.157,137.619,435.156,176.298,17.810,152.533
C06276=1094.152,137.370,435.176,176.296,17.808,152.534
C06277=1094.146,137.121,435.195,176.293,17.808,152.534
C06278=1094.140,136.872,435.215,176.290,17.807,152.534
C06279=1094.135,136.623,435.236,176.288,17.806,152.535
C06280=1094.129,136.374,435.256,176.285,17.806,152.535
C06281=1094.124,136.124,435.276,176.282,17.805,152.536
C06282=1094.118,135.876,435.296,176.279,17.804,152.536
C06283=1094.113,135.627,435.316,176.277,17.804,152.536
C06284=1094.107,135.378,435.336,176.274,17.803,152.537
C06285=1094.101,135.128,435.355,176.271,17.802,152.537
C06286=1094.096,134.879,435.376,176.268,17.801,152.537
C06287=1094.090,134.630,435.396,176.266,17.801,152.538
C06288=1094.085,134.381,435.416,176.263,17.800,152.538
C06289=1094.079,134.132,435.436,176.260,17.799,152.538
C06290=1094.073,133.883,435.456,176.258,17.799,152.539
C06291=1094.068,133.633,435.476,176.255,17.798,152.539
C06292=1094.062,133.384,435.495,176.252,17.797,152.539
C06293=1094.056,133.136,435.515,176.249,17.796,152.540
C06294=1094.051,132.886,435.535,176.248,17.796,152.540
C06295=1094.045,132.637,435.555,176.245,17.795,152.540
C06296=1094.040,132.387,435.575,176.242,17.794,152.541
C06297=1094.034,132.138,435.595,176.239,17.793,152.541
C06298=1094.028,131.889,435.614,176.237,17.793,152.542
C06299=1094.022,131.640,435.634,176.234,17.792,152.542
C06300=1094.016,131.391,435.654,176.231,17.791,152.542
C06301=1094.012,131.142,435.674,176.229,17.790,152.542
C06302=1094.006,130.893,435.694,176.226,17.789,152.543
C06303=1094.000,130.643,435.713,176.223,17.789,152.543
C06304=1093.994,130.395,435.733,176.220,17.788,152.544
C06305=1093.988,130.145,435.752,176.218,17.787,152.544
C06306=1093.982,129.896,435.772,176.215,17.787,152.544
C06307=1093.977,129.647,435.792,176.212,17.786,152.545
C06308=1093.971,129.398,435.812,176.210,17.785,152.545
C06309=1093.966,129.148,435.831,176.207,17.784,152.545
C06310=1093.960,128.900,435.851,176.205,17.783,152.546
C06311=1093.954,128.650,435.871,176.203,17.783,152.546
C06312=1093.948,128.401,435.891,176.200,17.782,152.546
C06313=1093.942,128.125,435.912,176.197,17.781,152.547
C06314=1093.936,127.849,435.934,176.194,17.780,152.547
C06315=1093.930,127.573,435.955,176.191,17.780,152.547
C06316=1093.923,127.298,435.977,176.188,17.779,152.548
C06317=1093.918,127.048,435.997,176.185,17.778,152.548
C06318=1093.912,126.799,436.016,176.183,17.777,152.549
C06319=1093.906,126.550,436.036,176.180,17.776,152.549
C06320=1093.900,126.301,436.055,176.177,17.776,152.549
C06321=1093.894,126.052,436.075,176.175,17.774,152.549
C06322=1093.889,125.802,436.095,176.172,17.774,152.550
C06323=1093.884,125.553,436.114,176.170,17.773,152.550
C06324=1093.878,125.304,436.134,176.167,17.772,152.551
C06325=1093.873,125.055,436.153,176.165,17.772,152.551
C06326=1093.867,124.806,436.172,176.162,17.771,152.551
C06327=1093.861,124.556,436.191,176.159,17.770,152.551
C06328=1093.855,124.307,436.211,176.157,17.769,152.552
C06329=1093.850,124.058,436.231,176.154,17.768,152.552
C06330=1093.845,123.809,436.249,176.151,17.767,152.552
C06331=1093.839,123.560,436.269,176.149,17.767,152.553
C06332=1093.833,123.311,436.289,176.147,17.766,152.553
C06333=1093.827,123.061,436.308,176.144,17.765,152.553
C06334=1093.821,122.812,436.327,176.141,17.764,152.554
C06335=1093.816,122.563,436.346,176.139,17.763,152.554
C06336=1093.810,122.314,436.366,176.136,17.762,152.554
C06337=1093.805,122.065,436.386,176.133,17.762,152.555
C06338=1093.800,121.815,436.405,176.131,17.761,152.555
C06339=1093.794,121.566,436.424,176.129,17.760,152.555
C06340=1093.788,121.316,436.444,176.126,17.759,152.556
C06341=1093.783,121.068,436.462,176.124,17.758,152.556
C06342=1093.777,120.819,436.482,176.121,17.757,152.556
C06343=1093.772,120.569,436.502,176.118,17.756,152.557
C06344=1093.766,120.320,436.521,176.116,17.756,152.557
C06345=1093.761,120.071,436.540,176.113,17.755,152.557
C06346=1093.755,119.822,436.559,176.111,17.753,152.557
C06347=1093.749,119.572,436.578,176.108,17.753,152.558
C06348=1093.744,119.323,436.597,176.106,17.752,152.558
C06349=1093.739,119.074,436.616,176.103,17.751,152.558
C06350=1093.733,118.825,436.636,176.101,17.750,152.558
C06351=1093.727,118.575,436.655,176.098,17.750,152.559
C06352=1093.721,118.326,436.673,176.095,17.748,152.559
C06353=1093.716,118.078,436.692,176.093,17.748,152.559
C06354=1093.710,117.829,436.712,176.091,17.747,152.560
C06355=1093.704,117.579,436.732,176.088,17.746,152.560
C06356=1093.699,117.331,436.750,176.086,17.745,152.560
C06357=1093.693,117.081,436.770,176.083,17.744,152.561
C06358=1093.688,116.831,436.788,176.080,17.743,152.561
C06359=1093.682,116.582,436.807,176.078,17.742,152.561
C06360=1093.677,116.333,436.826,176.076,17.741,152.561
C06361=1093.671,116.083,436.846,176.073,17.740,152.562
C06362=1093.666,115.834,436.865,176.071,17.740,152.562
C06363=1093.661,115.585,436.884,176.068,17.739,152.562
C06364=1093.655,115.336,436.903,176.065,17.737,152.563
C06365=1093.649,115.086,436.922,176.063,17.737,152.563
C06366=1093.644,114.838,436.941,176.061,17.736,152.563
C06367=1093.639,114.588,436.960,176.058,17.734,152.563
C06368=1093.632,114.339,436.979,176.056,17.734,152.564
C06369=1093.627,114.090,436.998,176.053,17.733,152.564
C06370=1093.621,113.841,437.017,176.050,17.732,152.564
C06371=1093.616,113.591,437.036,176.048,17.731,152.565
C06372=1093.610,113.343,437.054,176.046,17.730,152.565
C06373=1093.604,113.093,437.073,176.043,17.729,152.565
C06374=1093.599,112.844,437.092,176.041,17.729,152.565
C06375=1093.594,112.595,437.111,176.038,17.728,152.566
C06376=1093.587,112.346,437.130,176.035,17.726,152.566
C06377=1093.581,112.069,437.150,176.033,17.726,152.566
C06378=1093.575,111.793,437.172,176.031,17.725,152.567
C06379=1093.569,111.517,437.192,176.028,17.724,152.567
C06380=1093.563,111.242,437.213,176.025,17.723,152.567
C06381=1093.557,110.992,437.232,176.022,17.721,152.567
C06382=1093.551,110.743,437.251,176.020,17.720,152.568
C06383=1093.546,110.494,437.269,176.018,17.720,152.568
C06384=1093.540,110.244,437.288,176.015,17.718,152.568
C06385=1093.534,109.995,437.307,176.013,17.718,152.569
C06386=1093.529,109.746,437.326,176.010,17.717,152.569
C06387=1093.523,109.497,437.344,176.007,17.716,152.569
C06388=1093.518,109.248,437.363,176.005,17.715,152.569
C06389=1093.512,108.998,437.382,176.003,17.714,152.570
C06390=1093.506,108.749,437.400,176.000,17.713,152.570
C06391=1093.501,108.500,437.419,175.998,17.712,152.570
C06392=1093.494,108.251,437.437,175.995,17.711,152.571
C06393=1093.489,108.001,437.456,175.993,17.710,152.571
C06394=1093.484,107.752,437.475,175.991,17.709,152.571
C06395=1093.477,107.503,437.493,175.988,17.708,152.571
C06396=1093.473,107.254,437.511,175.986,17.708,152.572
C06397=1093.466,107.005,437.530,175.983,17.706,152.572
C06398=1093.460,106.755,437.549,175.981,17.705,152.572
C06399=1093.455,106.506,437.567,175.979,17.705,152.572
C06400=1093.449,106.257,437.586,175.976,17.703,152.573
C06401=1093.444,106.007,437.604,175.973,17.702,152.573
C06402=1093.438,105.758,437.623,175.971,17.702,152.573
C06403=1093.433,105.509,437.641,175.969,17.700,152.573
C06404=1093.427,105.260,437.660,175.967,17.700,152.574
C06405=1093.422,105.011,437.679,175.964,17.699,152.574
C06406=1093.416,104.761,437.697,175.961,17.697,152.574
C06407=1093.410,104.512,437.716,175.959,17.697,152.574
C06408=1093.404,104.263,437.733,175.957,17.696,152.575
C06409=1093.399,104.013,437.753,175.955,17.695,152.575
C06410=1093.393,103.764,437.770,175.952,17.694,152.575
C06411=1093.388,103.515,437.789,175.949,17.693,152.575
C06412=1093.382,103.266,437.807,175.947,17.692,152.576
C06413=1093.376,103.016,437.826,175.945,17.691,152.576
C06414=1093.371,102.767,437.844,175.942,17.690,152.576
C06415=1093.365,102.517,437.862,175.940,17.689,152.576
C06416=1093.360,102.269,437.881,175.938,17.687,152.577
C06417=1093.354,102.019,437.899,175.936,17.687,152.577
C06418=1093.348,101.770,437.917,175.933,17.686,152.577
C06419=1093.343,101.520,437.936,175.930,17.684,152.577
C06420=1093.337,101.272,437.954,175.928,17.684,152.578
C06421=1093.332,101.022,437.973,175.926,17.683,152.578
C06422=1093.326,100.773,437.990,175.924,17.682,152.578
C06423=1093.320,100.524,438.009,175.921,17.681,152.578
C06424=1093.315,100.274,438.027,175.918,17.680,152.579
C06425=1093.309,100.025,438.045,175.917,17.678,152.579
C06426=1093.303,99.776,438.063,175.914,17.677,152.579
C06427=1093.298,99.526,438.082,175.912,17.677,152.579
C06428=1093.292,99.277,438.099,175.909,17.675,152.580
C06429=1093.286,99.028,438.118,175.906,17.674,152.580
C06430=1093.281,98.779,438.136,175.905,17.674,152.580
C06431=1093.276,98.530,438.154,175.902,17.673,152.580
C06432=1093.269,98.280,438.172,175.900,17.672,152.581
C06433=1093.264,98.031,438.190,175.897,17.670,152.581
C06434=1093.258,97.781,438.209,175.895,17.669,152.581
C06435=1093.252,97.533,438.227,175.893,17.668,152.581
C06436=1093.246,97.283,438.245,175.890,17.667,152.582
C06437=1093.241,97.034,438.263,175.888,17.667,152.582
C06438=1093.235,96.784,438.281,175.886,17.665,152.582
C06439=1093.230,96.536,438.299,175.883,17.664,152.582
C06440=1093.223,96.286,438.317,175.881,17.663,152.582
C06441=1093.218,96.010,438.337,175.878,17.662,152.583
C06442=1093.212,95.735,438.357,175.876,17.661,152.583
C06443=1093.206,95.458,438.377,175.873,17.660,152.583
C06444=1093.199,95.182,438.397,175.870,17.658,152.583
C06445=1093.193,94.933,438.415,175.869,17.657,152.584
C06446=1093.188,94.684,438.432,175.866,17.656,152.584
C06447=1093.182,94.434,438.451,175.864,17.656,152.584
C06448=1093.176,94.185,438.469,175.861,17.654,152.584
C06449=1093.171,93.936,438.487,175.859,17.653,152.585
C06450=1093.165,93.686,438.505,175.857,17.652,152.585
C06451=1093.160,93.437,438.523,175.854,17.651,152.585
C06452=1093.155,93.188,438.540,175.852,17.650,152.585
C06453=1093.148,92.938,438.558,175.850,17.649,152.585
C06454=1093.143,92.689,438.576,175.848,17.648,152.586
C06455=1093.137,92.440,438.593,175.845,17.646,152.586
C06456=1093.132,92.190,438.612,175.843,17.645,152.586
C06457=1093.126,91.941,438.629,175.841,17.645,152.586
C06458=1093.121,91.692,438.647,175.838,17.643,152.586
C06459=1093.115,91.443,438.666,175.836,17.642,152.587
C06460=1093.109,91.194,438.683,175.834,17.641,152.587
C06461=1093.104,90.945,438.701,175.832,17.640,152.587
C06462=1093.098,90.695,438.719,175.829,17.639,152.587
C06463=1093.093,90.446,438.737,175.827,17.638,152.588
C06464=1093.086,90.196,438.755,175.825,17.636,152.588
C06465=1093.081,89.947,438.772,175.822,17.635,152.588
C06466=1093.075,89.698,438.790,175.820,17.635,152.588
C06467=1093.069,89.448,438.808,175.818,17.634,152.588
C06468=1093.064,89.199,438.825,175.816,17.632,152.589
C06469=1093.058,88.950,438.843,175.813,17.631,152.589
C06470=1093.052,88.700,438.860,175.810,17.630,152.589
C06471=1093.047,88.451,438.878,175.809,17.629,152.589
C06472=1093.041,88.202,438.895,175.806,17.628,152.589
C06473=1093.035,87.952,438.913,175.804,17.627,152.590
C06474=1093.030,87.703,438.931,175.802,17.625,152.590
C06475=1093.024,87.454,438.948,175.800,17.625,152.590
C06476=1093.018,87.204,438.966,175.797,17.623,152.590
C06477=1093.013,86.955,438.984,175.795,17.623,152.590
C06478=1093.007,86.706,439.002,175.793,17.621,152.591
C06479=1093.001,86.456,439.019,175.790,17.620,152.591
C06480=1092.995,86.208,439.036,175.788,17.619,152.591
C06481=1092.990,85.958,439.053,175.786,17.617,152.591
C06482=1092.984,85.709,439.071,175.784,17.617,152.591
C06483=1092.978,85.459,439.089,175.781,17.616,152.592
C06484=1092.972,85.210,439.106,175.780,17.615,152.592
C06485=1092.967,84.961,439.124,175.777,17.613,152.592
C06486=1092.962,84.711,439.141,175.775,17.612,152.592
C06487=1092.956,84.462,439.159,175.773,17.611,152.592
C06488=1092.950,84.213,439.176,175.770,17.609,152.593
C06489=1092.944,83.964,439.194,175.768,17.609,152.593
C06490=1092.939,83.715,439.211,175.766,17.607,152.593
C06491=1092.933,83.464,439.229,175.764,17.607,152.593
C06492=1092.928,83.215,439.246,175.761,17.605,152.593
C06493=1092.922,82.966,439.264,175.759,17.604,152.594
C06494=1092.917,82.717,439.281,175.757,17.603,152.594
C06495=1092.911,82.467,439.299,175.755,17.602,152.594
C06496=1092.905,82.218,439.315,175.753,17.600,152.594
C06497=1092.899,81.969,439.333,175.751,17.600,152.594
C06498=1092.894,81.719,439.350,175.748,17.598,152.594
C06499=1092.888,81.470,439.367,175.746,17.597,152.595
C06500=1092.883,81.221,439.385,175.744,17.596,152.595
C06501=1092.877,80.971,439.402,175.741,17.595,152.595
C06502=1092.871,80.722,439.420,175.740,17.593,152.595
C06503=1092.866,80.473,439.437,175.737,17.592,152.595
C06504=1092.861,80.223,439.454,175.735,17.591,152.596
C06505=1092.854,79.948,439.473,175.732,17.590,152.596
C06506=1092.848,79.672,439.492,175.730,17.588,152.596
C06507=1092.842,79.396,439.512,175.728,17.587,152.596
C06508=1092.835,79.119,439.531,175.726,17.586,152.596
C06509=1092.830,78.870,439.548,175.723,17.584,152.596
C06510=1092.824,78.621,439.565,175.720,17.583,152.597
C06511=1092.818,78.372,439.582,175.719,17.582,152.597
C06512=1092.813,78.123,439.600,175.716,17.581,152.597
C06513=1092.807,77.873,439.616,175.714,17.580,152.597
C06514=1092.801,77.623,439.634,175.712,17.578,152.597
C06515=1092.795,77.374,439.651,175.710,17.578,152.598
C06516=1092.790,77.125,439.668,175.708,17.576,152.598
C06517=1092.785,76.875,439.685,175.706,17.575,152.598
C06518=1092.778,76.627,439.702,175.703,17.574,152.598
C06519=1092.773,76.377,439.719,175.701,17.573,152.598
C06520=1092.768,76.128,439.736,175.699,17.571,152.598
C06521=1092.761,75.878,439.753,175.697,17.570,152.599
C06522=1092.755,75.629,439.771,175.695,17.569,152.599
C06523=1092.750,75.379,439.788,175.693,17.568,152.599
C06524=1092.744,75.131,439.805,175.690,17.567,152.599
C06525=1092.739,74.881,439.821,175.689,17.566,152.599
C06526=1092.733,74.632,439.839,175.686,17.564,152.599
C06527=1092.727,74.382,439.855,175.684,17.563,152.600
C06528=1092.722,74.133,439.873,175.682,17.562,152.600
C06529=1092.716,73.883,439.890,175.680,17.561,152.600
C06530=1092.710,73.634,439.906,175.677,17.559,152.600
C06531=1092.704,73.385,439.924,175.676,17.558,152.600
C06532=1092.699,73.135,439.941,175.673,17.557,152.600
C06533=1092.693,72.886,439.958,175.671,17.555,152.601
C06534=1092.688,72.637,439.974,175.669,17.554,152.601
C06535=1092.683,72.387,439.991,175.666,17.553,152.601
C06536=1092.676,72.138,440.008,175.665,17.552,152.601
C06537=1092.671,71.889,440.025,175.662,17.550,152.601
C06538=1092.665,71.639,440.041,175.660,17.549,152.601
C06539=1092.660,71.390,440.059,175.658,17.548,152.602
C06540=1092.654,71.141,440.075,175.656,17.547,152.602
C06541=1092.648,70.891,440.092,175.654,17.545,152.602
C06542=1092.642,70.641,440.110,175.652,17.544,152.602
C06543=1092.636,70.392,440.126,175.649,17.543,152.602
C06544=1092.631,70.142,440.143,175.648,17.542,152.602
C06545=1092.625,69.894,440.160,175.645,17.540,152.602
C06546=1092.620,69.644,440.177,175.644,17.539,152.603
C06547=1092.614,69.395,440.193,175.641,17.538,152.603
C06548=1092.609,69.145,440.210,175.639,17.537,152.603
C06549=1092.602,68.896,440.227,175.637,17.535,152.603
C06550=1092.597,68.647,440.244,175.635,17.535,152.603
C06551=1092.591,68.397,440.260,175.632,17.533,152.603
C06552=1092.586,68.148,440.277,175.631,17.532,152.603
C06553=1092.580,67.899,440.294,175.628,17.530,152.604
C06554=1092.574,67.649,440.311,175.626,17.530,152.604
C06555=1092.569,67.400,440.327,175.624,17.528,152.604
C06556=1092.563,67.150,440.344,175.622,17.527,152.604
C06557=1092.557,66.901,440.360,175.620,17.525,152.604
C06558=1092.551,66.652,440.376,175.618,17.525,152.604
C06559=1092.546,66.403,440.394,175.615,17.523,152.605
C06560=1092.540,66.153,440.410,175.614,17.522,152.605
C06561=1092.535,65.904,440.427,175.612,17.521,152.605
C06562=1092.529,65.654,440.443,175.610,17.519,152.605
C06563=1092.523,65.405,440.460,175.608,17.518,152.605
C06564=1092.518,65.155,440.476,175.605,17.517,152.605
C06565=1092.512,64.906,440.493,175.604,17.516,152.605
C06566=1092.506,64.657,440.510,175.601,17.514,152.605
C06567=1092.500,64.407,440.527,175.600,17.513,152.606
C06568=1092.494,64.158,440.543,175.597,17.512,152.606
C06569=1092.486,63.793,440.568,175.594,17.510,152.606
C06570=1092.478,63.428,440.591,175.591,17.508,152.606
C06571=1092.469,63.063,440.615,175.588,17.506,152.607
C06572=1092.460,62.698,440.639,175.585,17.504,152.607
C06573=1092.455,62.448,440.656,175.583,17.503,152.607
C06574=1092.449,62.199,440.672,175.581,17.502,152.607
C06575=1092.443,61.949,440.688,175.578,17.500,152.607
C06576=1092.437,61.700,440.705,175.577,17.499,152.607
C06577=1092.431,61.451,440.721,175.574,17.498,152.607
C06578=1092.426,61.201,440.738,175.573,17.497,152.607
C06579=1092.420,60.952,440.754,175.570,17.495,152.608
C06580=1092.414,60.702,440.770,175.568,17.494,152.608
C06581=1092.408,60.453,440.786,175.566,17.493,152.608
C06582=1092.402,60.204,440.803,175.564,17.492,152.608
C06583=1092.397,59.955,440.819,175.563,17.490,152.608
C06584=1092.392,59.705,440.835,175.560,17.489,152.608
C06585=1092.386,59.456,440.852,175.558,17.488,152.608
C06586=1092.380,59.207,440.868,175.556,17.487,152.609
C06587=1092.374,58.957,440.884,175.554,17.485,152.609
C06588=1092.368,58.708,440.900,175.552,17.484,152.609
C06589=1092.363,58.458,440.917,175.550,17.483,152.609
C06590=1092.357,58.208,440.933,175.548,17.481,152.609
C06591=1092.351,57.959,440.949,175.546,17.480,152.609
C06592=1092.345,57.710,440.965,175.543,17.478,152.609
C06593=1092.339,57.460,440.982,175.542,17.477,152.609
C06594=1092.333,57.211,440.998,175.539,17.476,152.610
C06595=1092.328,56.962,441.014,175.537,17.475,152.610
C06596=1092.322,56.713,441.031,175.536,17.474,152.610
C06597=1092.317,56.463,441.046,175.533,17.472,152.610
C06598=1092.311,56.213,441.062,175.532,17.471,152.610
C06599=1092.305,55.964,441.079,175.529,17.469,152.610
C06600=1092.299,55.715,441.095,175.528,17.468,152.610
C06601=1092.293,55.465,441.111,175.525,17.467,152.611
C06602=1092.287,55.215,441.127,175.524,17.465,152.611
C06603=1092.282,54.967,441.143,175.521,17.464,152.611
C06604=1092.277,54.717,441.159,175.520,17.463,152.611
C06605=1092.271,54.468,441.176,175.517,17.461,152.611
C06606=1092.265,54.218,441.192,175.515,17.460,152.611
C06607=1092.259,53.968,441.207,175.514,17.459,152.611
C06608=1092.253,53.719,441.224,175.511,17.457,152.611
C06609=1092.248,53.470,441.240,175.510,17.456,152.611
C06610=1092.242,53.220,441.255,175.507,17.454,152.612
C06611=1092.236,52.971,441.271,175.506,17.453,152.612
C06612=1092.230,52.722,441.288,175.503,17.452,152.612
C06613=1092.224,52.472,441.304,175.502,17.450,152.612
C06614=1092.219,52.223,441.319,175.499,17.449,152.612
C06615=1092.214,51.973,441.336,175.497,17.448,152.612
C06616=1092.208,51.724,441.352,175.496,17.447,152.612
C06617=1092.203,51.474,441.368,175.493,17.445,152.612
C06618=1092.197,51.225,441.384,175.492,17.444,152.612
C06619=1092.191,50.976,441.400,175.489,17.442,152.613
C06620=1092.186,50.726,441.415,175.488,17.441,152.613
C06621=1092.180,50.477,441.432,175.485,17.439,152.613
C06622=1092.174,50.227,441.447,175.484,17.438,152.613
C06623=1092.169,49.978,441.463,175.482,17.437,152.613
C06624=1092.163,49.729,441.479,175.479,17.435,152.613
C06625=1092.153,49.319,441.505,175.476,17.433,152.613
C06626=1092.144,48.909,441.531,175.473,17.431,152.613
C06627=1092.135,48.499,441.558,175.470,17.428,152.613
C06628=1092.126,48.090,441.583,175.467,17.426,152.614
C06629=1092.119,47.813,441.601,175.464,17.424,152.614
C06630=1092.113,47.537,441.618,175.463,17.423,152.614
C06631=1092.107,47.260,441.636,175.460,17.422,152.614
C06632=1092.101,46.984,441.653,175.458,17.420,152.614
C06633=1092.095,46.735,441.669,175.456,17.419,152.614
C06634=1092.089,46.485,441.685,175.454,17.417,152.614
C06635=1092.084,46.236,441.701,175.452,17.416,152.614
C06636=1092.078,45.987,441.716,175.451,17.415,152.614
C06637=1092.072,45.737,441.732,175.448,17.413,152.615
C06638=1092.067,45.488,441.747,175.446,17.412,152.615
C06639=1092.061,45.239,441.764,175.444,17.410,152.615
C06640=1092.056,44.989,441.779,175.442,17.409,152.615
C06641=1092.050,44.740,441.795,175.440,17.407,152.615
C06642=1092.045,44.490,441.811,175.439,17.406,152.615
C06643=1092.039,44.240,441.826,175.437,17.405,152.615
C06644=1092.034,43.991,441.842,175.434,17.403,152.615
C06645=1092.028,43.741,441.858,175.433,17.402,152.615
C06646=1092.021,43.492,441.873,175.430,17.400,152.615
C06647=1092.016,43.243,441.889,175.429,17.399,152.616
C06648=1092.011,42.993,441.904,175.427,17.398,152.615
C06649=1092.005,42.744,441.920,175.425,17.396,152.616
C06650=1092.000,42.494,441.935,175.423,17.395,152.616
C06651=1091.993,42.245,441.950,175.421,17.393,152.616
C06652=1091.987,41.995,441.967,175.419,17.392,152.616
C06653=1091.982,41.746,441.982,175.418,17.391,152.616
C06654=1091.977,41.496,441.997,175.415,17.389,152.616
C06655=1091.971,41.247,442.014,175.414,17.388,152.616
C06656=1091.965,40.998,442.028,175.411,17.386,152.616
C06657=1091.959,40.748,442.044,175.410,17.385,152.616
C06658=1091.953,40.499,442.060,175.408,17.384,152.616
C06659=1091.948,40.249,442.075,175.406,17.382,152.617
C06660=1091.942,40.000,442.090,175.404,17.381,152.617
C06661=1091.937,39.751,442.106,175.402,17.379,152.617
C06662=1091.931,39.501,442.122,175.400,17.378,152.617
C06663=1091.925,39.251,442.137,175.399,17.377,152.617
C06664=1091.920,39.002,442.152,175.396,17.375,152.617
C06665=1091.914,38.753,442.168,175.394,17.374,152.617
C06666=1091.909,38.504,442.183,175.392,17.372,152.617
C06667=1091.903,38.254,442.199,175.391,17.371,152.617
C06668=1091.897,38.004,442.214,175.389,17.369,152.617
C06669=1091.892,37.755,442.229,175.387,17.368,152.617
C06670=1091.886,37.505,442.245,175.385,17.367,152.617
C06671=1091.879,37.256,442.260,175.383,17.365,152.617
C06672=1091.874,37.006,442.275,175.381,17.363,152.618
C06673=1091.868,36.757,442.290,175.379,17.362,152.618
C06674=1091.863,36.507,442.305,175.377,17.361,152.618
C06675=1091.856,36.258,442.321,175.375,17.360,152.618
C06676=1091.850,36.008,442.337,175.373,17.358,152.618
C06677=1091.845,35.759,442.352,175.372,17.356,152.618
C06678=1091.839,35.510,442.367,175.370,17.355,152.618
C06679=1091.834,35.260,442.382,175.367,17.353,152.618
C06680=1091.828,35.011,442.397,175.366,17.352,152.618
C06681=1091.822,34.761,442.412,175.364,17.351,152.618
C06682=1091.816,34.512,442.427,175.362,17.349,152.618
C06683=1091.810,34.262,442.443,175.360,17.348,152.618
C06684=1091.805,34.013,442.458,175.358,17.346,152.619
C06685=1091.799,33.763,442.473,175.356,17.345,152.619
C06686=1091.794,33.514,442.488,175.355,17.344,152.619
C06687=1091.787,33.264,442.503,175.352,17.342,152.619
C06688=1091.782,33.015,442.519,175.351,17.341,152.619
C06689=1091.776,32.766,442.533,175.348,17.339,152.619
C06690=1091.770,32.516,442.549,175.347,17.338,152.619
C06691=1091.764,32.267,442.564,175.345,17.336,152.619
C06692=1091.759,32.017,442.579,175.343,17.335,152.619
C06693=1091.752,31.741,442.596,175.341,17.334,152.619
C06694=1091.746,31.464,442.612,175.339,17.332,152.619
C06695=1091.740,31.189,442.629,175.338,17.330,152.619
C06696=1091.734,30.912,442.646,175.335,17.329,152.620
C06697=1091.728,30.663,442.660,175.334,17.327,152.619
C06698=1091.722,30.413,442.676,175.331,17.326,152.620
C06699=1091.716,30.164,442.690,175.330,17.324,152.620
C06700=1091.711,29.914,442.706,175.327,17.323,152.620
C06701=1091.705,29.665,442.721,175.326,17.321,152.620
C06702=1091.699,29.415,442.736,175.324,17.320,152.620
C06703=1091.694,29.166,442.751,175.322,17.318,152.620
C06704=1091.688,28.916,442.766,175.320,17.317,152.620
C06705=1091.682,28.667,442.781,175.319,17.316,152.620
C06706=1091.676,28.417,442.796,175.316,17.314,152.620
C06707=1091.671,28.168,442.811,175.315,17.313,152.620
C06708=1091.664,27.918,442.826,175.313,17.311,152.620
C06709=1091.659,27.669,442.841,175.311,17.310,152.620
C06710=1091.653,27.419,442.856,175.309,17.309,152.620
C06711=1091.647,27.170,442.870,175.307,17.306,152.620
C06712=1091.642,26.920,442.885,175.305,17.305,152.621
C06713=1091.636,26.671,442.900,175.304,17.304,152.621
C06714=1091.630,26.422,442.915,175.301,17.302,152.621
C06715=1091.625,26.172,442.930,175.300,17.301,152.621
C06716=1091.619,25.923,442.945,175.298,17.300,152.621
C06717=1091.613,25.673,442.959,175.296,17.298,152.621
C06718=1091.608,25.424,442.974,175.295,17.297,152.621
C06719=1091.601,25.174,442.989,175.293,17.295,152.621
C06720=1091.596,24.925,443.004,175.290,17.294,152.621
C06721=1091.590,24.675,443.019,175.289,17.293,152.621
C06722=1091.584,24.425,443.033,175.287,17.291,152.621
C06723=1091.578,24.176,443.048,175.285,17.289,152.621
C06724=1091.572,23.927,443.063,175.283,17.288,152.621
C06725=1091.567,23.677,443.078,175.282,17.287,152.621
C06726=1091.561,23.428,443.093,175.280,17.285,152.622
C06727=1091.555,23.178,443.107,175.278,17.284,152.622
C06728=1091.550,22.928,443.122,175.277,17.282,152.622
C06729=1091.544,22.679,443.137,175.274,17.281,152.622
C06730=1091.538,22.429,443.151,175.272,17.280,152.622
C06731=1091.532,22.180,443.166,175.271,17.278,152.622
C06732=1091.527,21.931,443.181,175.269,17.276,152.622
C06733=1091.521,21.681,443.196,175.267,17.275,152.622
C06734=1091.515,21.432,443.209,175.266,17.274,152.622
C06735=1091.509,21.182,443.224,175.263,17.272,152.622
C06736=1091.504,20.933,443.240,175.262,17.270,152.622
C06737=1091.498,20.683,443.253,175.260,17.269,152.622
C06738=1091.492,20.433,443.268,175.258,17.267,152.622
C06739=1091.486,20.185,443.283,175.256,17.266,152.622
C06740=1091.481,19.934,443.298,175.255,17.265,152.622
C06741=1091.475,19.685,443.312,175.252,17.263,152.622
C06742=1091.470,19.435,443.326,175.251,17.261,152.622
C06743=1091.463,19.186,443.341,175.249,17.260,152.622
C06744=1091.457,18.937,443.356,175.247,17.259,152.623
C06745=1091.452,18.687,443.370,175.246,17.257,152.623
C06746=1091.446,18.437,443.385,175.244,17.256,152.623
C06747=1091.441,18.188,443.399,175.241,17.254,152.623
C06748=1091.434,17.938,443.414,175.240,17.253,152.623
C06749=1091.429,17.689,443.429,175.238,17.252,152.623
C06750=1091.423,17.439,443.442,175.236,17.249,152.623
C06751=1091.417,17.190,443.457,175.235,17.248,152.623
C06752=1091.411,16.940,443.471,175.233,17.247,152.623
C06753=1091.405,16.691,443.486,175.231,17.245,152.623
C06754=1091.400,16.441,443.501,175.229,17.244,152.623
C06755=1091.394,16.192,443.515,175.228,17.243,152.623
C06756=1091.389,15.942,443.529,175.225,17.241,152.623
C06757=1091.382,15.667,443.545,175.224,17.240,152.623
C06758=1091.376,15.392,443.561,175.222,17.237,152.623
C06759=1091.369,15.118,443.577,175.220,17.236,152.623
C06760=1091.363,14.843,443.593,175.218,17.234,152.623
C06761=1091.358,14.594,443.607,175.216,17.233,152.623
C06762=1091.351,14.344,443.622,175.215,17.232,152.624
C06763=1091.346,14.094,443.636,175.212,17.230,152.624
C06764=1091.340,13.845,443.650,175.211,17.229,152.624
C06765=1091.334,13.595,443.664,175.209,17.228,152.624
C06766=1091.328,13.346,443.679,175.207,17.225,152.624
C06767=1091.323,13.097,443.693,175.205,17.224,152.624
C06768=1091.316,12.847,443.708,175.204,17.223,152.624
C06769=1091.311,12.597,443.722,175.202,17.222,152.624
C06770=1091.305,12.348,443.736,175.200,17.220,152.624
C06771=1091.298,12.098,443.750,175.199,17.218,152.624
C06772=1091.293,11.849,443.764,175.197,17.217,152.624
C06773=1091.287,11.600,443.778,175.194,17.216,152.624
C06774=1091.281,11.350,443.793,175.193,17.214,152.624
C06775=1091.275,11.100,443.806,175.191,17.213,152.624
C06776=1091.270,10.851,443.821,175.190,17.212,152.624
C06777=1091.264,10.601,443.835,175.188,17.210,152.624
C06778=1091.258,10.351,443.849,175.186,17.208,152.624
C06779=1091.252,10.102,443.864,175.185,17.207,152.624
C06780=1091.247,9.853,443.878,175.182,17.205,152.625
C06781=1091.240,9.603,443.892,175.181,17.204,152.625
C06782=1091.234,9.354,443.906,175.179,17.202,152.625
C06783=1091.229,9.104,443.920,175.177,17.201,152.625
C06784=1091.223,8.854,443.934,175.175,17.199,152.625
C06785=1091.217,8.605,443.948,175.174,17.198,152.625
C06786=1091.211,8.355,443.962,175.172,17.197,152.625
C06787=1091.206,8.106,443.976,175.170,17.195,152.625
C06788=1091.200,7.856,443.991,175.168,17.194,152.625
C06789=1091.193,7.607,444.004,175.167,17.192,152.625
C06790=1091.188,7.357,444.018,175.165,17.190,152.625
C06791=1091.182,7.108,444.032,175.163,17.189,152.625
C06792=1091.176,6.858,444.047,175.162,17.188,152.625
C06793=1091.171,6.609,444.061,175.160,17.187,152.625
C06794=1091.165,6.359,444.075,175.158,17.184,152.625
C06795=1091.160,6.109,444.089,175.156,17.183,152.625
C06796=1091.153,5.860,444.102,175.155,17.182,152.625
C06797=1091.147,5.611,444.117,175.153,17.181,152.625
C06798=1091.142,5.361,444.131,175.151,17.179,152.625
C06799=1091.136,5.111,444.145,175.149,17.177,152.625
C06800=1091.131,4.862,444.159,175.148,17.176,152.626
C06801=1091.125,4.612,444.172,175.146,17.174,152.626
C06802=1091.118,4.363,444.187,175.144,17.173,152.626
C06803=1091.113,4.113,444.201,175.143,17.171,152.626
C06804=1091.107,3.864,444.214,175.141,17.170,152.626
C06805=1091.102,3.614,444.228,175.139,17.168,152.626
C06806=1091.096,3.365,444.242,175.137,17.167,152.626
C06807=1091.090,3.115,444.255,175.136,17.165,152.626
C06808=1091.084,2.865,444.270,175.134,17.164,152.626
C06809=1091.078,2.615,444.284,175.132,17.162,152.626
C06810=1091.073,2.366,444.298,175.130,17.161,152.626
C06811=1091.067,2.117,444.312,175.129,17.160,152.626
C06812=1091.061,1.868,444.325,175.127,17.158,152.626
C06813=1091.055,1.618,444.339,175.125,17.157,152.626
C06814=1091.050,1.369,444.353,175.124,17.155,152.626
C06815=1091.044,1.118,444.367,175.122,17.154,152.626
C06816=1091.038,0.869,444.380,175.120,17.152,152.626
C06817=1091.032,0.619,444.394,175.118,17.151,152.626
C06818=1091.027,0.370,444.408,175.117,17.149,152.626
C06819=1091.021,0.120,444.422,175.115,17.148,152.626
C06820=1091.015,-0.129,444.435,175.113,17.146,152.626
C06821=1091.009,-0.402,444.451,175.111,17.145,152.626
C06822=1091.002,-0.675,444.466,175.109,17.142,152.626
C06823=1090.997,-0.947,444.481,175.108,17.141,152.626
C06824=1090.990,-1.221,444.496,175.105,17.139,152.626
C06825=1090.984,-1.470,444.510,175.104,17.138,152.626
C06826=1090.979,-1.720,444.523,175.102,17.136,152.626
C06827=1090.973,-1.969,444.537,175.101,17.135,152.626
C06828=1090.967,-2.218,444.551,175.099,17.133,152.627
C06829=1090.962,-2.468,444.564,175.097,17.132,152.627
C06830=1090.956,-2.718,444.578,175.096,17.130,152.627
C06831=1090.950,-2.967,444.592,175.094,17.129,152.627
C06832=1090.945,-3.216,444.605,175.092,17.127,152.627
C06833=1090.939,-3.466,444.619,175.090,17.126,152.627
C06834=1090.933,-3.715,444.633,175.089,17.124,152.627
C06835=1090.927,-3.966,444.647,175.087,17.123,152.627
C06836=1090.921,-4.215,444.660,175.085,17.121,152.627
C06837=1090.916,-4.465,444.673,175.083,17.120,152.627
C06838=1090.909,-4.714,444.686,175.082,17.118,152.627
C06839=1090.904,-4.964,444.700,175.080,17.117,152.627
C06840=1090.898,-5.213,444.714,175.079,17.116,152.627
C06841=1090.892,-5.463,444.727,175.077,17.114,152.627
C06842=1090.886,-5.712,444.741,175.075,17.113,152.627
C06843=1090.880,-5.962,444.755,175.074,17.111,152.627
C06844=1090.874,-6.212,444.768,175.072,17.110,152.627
C06845=1090.868,-6.462,444.781,175.070,17.108,152.627
C06846=1090.862,-6.711,444.795,175.068,17.107,152.627
C06847=1090.857,-6.961,444.809,175.067,17.105,152.627
C06848=1090.851,-7.210,444.822,175.065,17.104,152.627
C06849=1090.845,-7.459,444.836,175.063,17.102,152.627
C06850=1090.839,-7.709,444.849,175.061,17.101,152.627
C06851=1090.834,-7.959,444.862,175.060,17.099,152.627
C06852=1090.827,-8.208,444.875,175.058,17.098,152.628
C06853=1090.822,-8.458,444.889,175.057,17.097,152.627
C06854=1090.816,-8.707,444.902,175.055,17.095,152.628
C06855=1090.811,-8.957,444.916,175.053,17.094,152.628
C06856=1090.804,-9.206,444.929,175.052,17.092,152.628
C06857=1090.798,-9.456,444.942,175.050,17.091,152.628
C06858=1090.793,-9.705,444.956,175.048,17.089,152.628
C06859=1090.787,-9.955,444.969,175.046,17.088,152.628
C06860=1090.781,-10.205,444.982,175.045,17.086,152.628
C06861=1090.775,-10.454,444.996,175.043,17.085,152.628
C06862=1090.770,-10.704,445.010,175.042,17.084,152.628
C06863=1090.764,-10.953,445.022,175.039,17.082,152.628
C06864=1090.758,-11.203,445.036,175.038,17.080,152.628
C06865=1090.752,-11.452,445.049,175.036,17.079,152.628
C06866=1090.746,-11.702,445.062,175.035,17.078,152.628
C06867=1090.741,-11.952,445.076,175.033,17.076,152.628
C06868=1090.734,-12.201,445.089,175.031,17.074,152.628
C06869=1090.729,-12.451,445.102,175.030,17.073,152.628
C06870=1090.723,-12.700,445.115,175.028,17.072,152.628
C06871=1090.717,-12.950,445.129,175.027,17.070,152.628
C06872=1090.712,-13.200,445.142,175.025,17.068,152.628
C06873=1090.705,-13.449,445.155,175.023,17.067,152.628
C06874=1090.700,-13.699,445.169,175.022,17.066,152.628
C06875=1090.694,-13.949,445.181,175.020,17.064,152.628
C06876=1090.688,-14.198,445.195,175.019,17.063,152.628
C06877=1090.683,-14.448,445.208,175.016,17.061,152.628
C06878=1090.676,-14.697,445.221,175.015,17.060,152.628
C06879=1090.671,-14.947,445.235,175.013,17.058,152.629
C06880=1090.665,-15.197,445.248,175.012,17.057,152.628
C06881=1090.659,-15.446,445.261,175.010,17.056,152.629
C06882=1090.653,-15.696,445.273,175.008,17.054,152.629
C06883=1090.647,-15.946,445.287,175.006,17.052,152.629
C06884=1090.642,-16.195,445.300,175.005,17.051,152.629
C06885=1090.635,-16.466,445.314,175.003,17.050,152.629
C06886=1090.629,-16.738,445.328,175.001,17.048,152.629
C06887=1090.622,-17.009,445.342,175.000,17.046,152.629
C06888=1090.616,-17.280,445.356,174.997,17.045,152.629
C06889=1090.610,-17.528,445.369,174.996,17.043,152.629
C06890=1090.605,-17.779,445.382,174.994,17.042,152.629
C06891=1090.599,-18.028,445.396,174.993,17.040,152.629
C06892=1090.593,-18.278,445.408,174.991,17.039,152.629
C06893=1090.587,-18.527,445.422,174.990,17.038,152.629
C06894=1090.581,-18.777,445.434,174.987,17.036,152.629
C06895=1090.575,-19.026,445.448,174.986,17.035,152.629
C06896=1090.569,-19.276,445.461,174.984,17.033,152.629
C06897=1090.563,-19.526,445.474,174.983,17.032,152.629
C06898=1090.557,-19.775,445.486,174.981,17.031,152.629
C06899=1090.551,-20.025,445.500,174.979,17.029,152.629
C06900=1090.545,-20.275,445.512,174.978,17.027,152.629
C06901=1090.540,-20.524,445.526,174.976,17.026,152.629
C06902=1090.534,-20.773,445.538,174.975,17.025,152.629
C06903=1090.528,-21.023,445.551,174.973,17.024,152.630
C06904=1090.522,-21.273,445.564,174.972,17.022,152.629
C06905=1090.516,-21.522,445.577,174.969,17.020,152.630
C06906=1090.510,-21.772,445.590,174.968,17.019,152.630
C06907=1090.505,-22.022,445.603,174.966,17.018,152.630
C06908=1090.499,-22.272,445.616,174.965,17.016,152.630
C06909=1090.493,-22.521,445.629,174.963,17.015,152.630
C06910=1090.488,-22.770,445.641,174.961,17.013,152.630
C06911=1090.482,-23.020,445.654,174.959,17.012,152.630
C06912=1090.475,-23.269,445.667,174.958,17.010,152.630
C06913=1090.469,-23.519,445.679,174.956,17.009,152.630
C06914=1090.464,-23.769,445.693,174.955,17.008,152.630
C06915=1090.458,-24.019,445.706,174.953,17.006,152.630
C06916=1090.452,-24.269,445.718,174.951,17.004,152.630
C06917=1090.447,-24.518,445.731,174.950,17.003,152.630
C06918=1090.441,-24.767,445.744,174.948,17.002,152.630
C06919=1090.435,-25.017,445.756,174.947,17.000,152.630
C06920=1090.429,-25.267,445.769,174.945,16.999,152.630
C06921=1090.423,-25.516,445.782,174.944,16.997,152.630
C06922=1090.418,-25.766,445.795,174.941,16.996,152.630
C06923=1090.412,-26.015,445.808,174.940,16.995,152.630
C06924=1090.406,-26.265,445.820,174.938,16.993,152.630
C06925=1090.400,-26.515,445.833,174.937,16.992,152.630
C06926=1090.394,-26.764,445.846,174.935,16.990,152.630
C06927=1090.389,-27.014,445.858,174.934,16.989,152.631
C06928=1090.383,-27.264,445.871,174.932,16.988,152.630
C06929=1090.377,-27.513,445.884,174.930,16.986,152.631
C06930=1090.371,-27.763,445.897,174.929,16.984,152.631
C06931=1090.365,-28.013,445.909,174.927,16.983,152.631
C06932=1090.359,-28.262,445.922,174.925,16.982,152.631
C06933=1090.353,-28.511,445.935,174.924,16.980,152.631
C06934=1090.347,-28.761,445.947,174.922,16.979,152.631
C06935=1090.341,-29.010,445.959,174.921,16.978,152.631
C06936=1090.335,-29.260,445.972,174.919,16.976,152.631
C06937=1090.329,-29.510,445.984,174.917,16.975,152.631
C06938=1090.323,-29.760,445.997,174.916,16.973,152.631
C06939=1090.317,-30.009,446.010,174.914,16.972,152.631
C06940=1090.312,-30.259,446.022,174.913,16.971,152.631
C06941=1090.306,-30.508,446.035,174.911,16.969,152.631
C06942=1090.300,-30.758,446.047,174.910,16.968,152.631
C06943=1090.294,-31.008,446.060,174.907,16.966,152.631
C06944=1090.289,-31.257,446.072,174.906,16.965,152.631
C06945=1090.283,-31.507,446.085,174.904,16.963,152.631
C06946=1090.276,-31.756,446.097,174.903,16.962,152.631
C06947=1090.270,-32.006,446.110,174.901,16.961,152.631
C06948=1090.264,-32.255,446.122,174.900,16.960,152.631
C06949=1090.258,-32.526,446.136,174.897,16.958,152.632
C06950=1090.252,-32.797,446.150,174.896,16.956,152.632
C06951=1090.245,-33.067,446.163,174.894,16.955,152.632
C06952=1090.239,-33.337,446.176,174.893,16.954,152.632
C06953=1090.233,-33.587,446.189,174.890,16.952,152.632
C06954=1090.228,-33.836,446.201,174.889,16.950,152.632
C06955=1090.221,-34.085,446.213,174.887,16.949,152.632
C06956=1090.215,-34.335,446.226,174.886,16.948,152.632
C06957=1090.209,-34.585,446.238,174.884,16.947,152.632
C06958=1090.204,-34.834,446.250,174.883,16.945,152.632
C06959=1090.198,-35.084,446.263,174.881,16.944,152.632
C06960=1090.192,-35.334,446.275,174.880,16.943,152.632
C06961=1090.187,-35.583,446.288,174.878,16.941,152.632
C06962=1090.180,-35.833,446.300,174.876,16.939,152.632
C06963=1090.174,-36.083,446.312,174.874,16.938,152.632
C06964=1090.168,-36.333,446.325,174.873,16.937,152.632
C06965=1090.163,-36.582,446.337,174.871,16.936,152.632
C06966=1090.157,-36.832,446.349,174.870,16.934,152.632
C06967=1090.151,-37.082,446.362,174.868,16.933,152.632
C06968=1090.145,-37.331,446.374,174.867,16.931,152.632
C06969=1090.139,-37.580,446.386,174.865,16.930,152.632
C06970=1090.133,-37.830,446.399,174.863,16.928,152.633
C06971=1090.128,-38.079,446.411,174.862,16.927,152.632
C06972=1090.123,-38.330,446.423,174.860,16.926,152.633
C06973=1090.116,-38.580,446.435,174.859,16.924,152.633
C06974=1090.111,-38.829,446.447,174.857,16.923,152.633
C06975=1090.105,-39.079,446.459,174.855,16.922,152.633
C06976=1090.098,-39.328,446.471,174.854,16.920,152.633
C06977=1090.093,-39.577,446.484,174.852,16.919,152.633
C06978=1090.087,-39.827,446.496,174.851,16.918,152.633
C06979=1090.080,-40.077,446.508,174.849,16.916,152.633
C06980=1090.075,-40.326,446.520,174.847,16.915,152.633
C06981=1090.069,-40.576,446.533,174.845,16.914,152.633
C06982=1090.063,-40.826,446.544,174.844,16.912,152.633
C06983=1090.057,-41.076,446.557,174.842,16.911,152.633
C06984=1090.051,-41.325,446.569,174.841,16.909,152.633
C06985=1090.045,-41.575,446.581,174.839,16.908,152.633
C06986=1090.039,-41.825,446.593,174.838,16.907,152.633
C06987=1090.033,-42.073,446.605,174.836,16.905,152.633
C06988=1090.027,-42.324,446.617,174.835,16.904,152.633
C06989=1090.021,-42.574,446.629,174.833,16.903,152.633
C06990=1090.015,-42.823,446.641,174.831,16.901,152.633
C06991=1090.009,-43.073,446.653,174.829,16.900,152.634
C06992=1090.004,-43.322,446.666,174.828,16.899,152.634
C06993=1089.998,-43.572,446.677,174.826,16.897,152.634
C06994=1089.992,-43.822,446.689,174.825,16.896,152.634
C06995=1089.986,-44.071,446.701,174.823,16.895,152.634
C06996=1089.980,-44.321,446.714,174.822,16.893,152.634
C06997=1089.974,-44.571,446.726,174.820,16.892,152.634
C06998=1089.968,-44.820,446.737,174.819,16.891,152.634
C06999=1089.962,-45.070,446.750,174.817,16.890,152.634
C07000=1089.956,-45.319,446.761,174.816,16.888,152.634
C07001=1089.951,-45.569,446.773,174.814,16.887,152.634
C07002=1089.945,-45.819,446.786,174.813,16.886,152.634
C07003=1089.939,-46.068,446.797,174.810,16.884,152.634
C07004=1089.933,-46.318,446.810,174.809,16.883,152.634
C07005=1089.927,-46.567,446.821,174.807,16.881,152.634
C07006=1089.921,-46.817,446.833,174.806,16.880,152.634
C07007=1089.914,-47.067,446.845,174.804,16.879,152.635
C07008=1089.909,-47.317,446.857,174.803,16.877,152.635
C07009=1089.903,-47.566,446.868,174.801,16.876,152.635
C07010=1089.898,-47.815,446.881,174.799,16.875,152.635
C07011=1089.892,-48.066,446.892,174.798,16.874,152.635
C07012=1089.886,-48.315,446.904,174.796,16.873,152.635
C07013=1089.880,-48.586,446.917,174.795,16.871,152.635
C07014=1089.873,-48.856,446.930,174.793,16.869,152.635
C07015=1089.866,-49.127,446.943,174.791,16.868,152.635
C07016=1089.861,-49.398,446.956,174.790,16.867,152.635
C07017=1089.854,-49.648,446.968,174.788,16.865,152.635
C07018=1089.849,-49.897,446.979,174.786,16.864,152.635
C07019=1089.842,-50.147,446.991,174.785,16.863,152.635
C07020=1089.837,-50.396,447.003,174.783,16.862,152.635
C07021=1089.831,-50.646,447.014,174.782,16.860,152.635
C07022=1089.825,-50.895,447.027,174.780,16.859,152.635
C07023=1089.819,-51.146,447.038,174.779,16.858,152.635
C07024=1089.812,-51.395,447.050,174.777,16.857,152.635
C07025=1089.806,-51.644,447.061,174.775,16.856,152.636
C07026=1089.801,-51.895,447.073,174.774,16.854,152.636
C07027=1089.795,-52.143,447.085,174.772,16.852,152.636
C07028=1089.788,-52.394,447.096,174.770,16.851,152.636
C07029=1089.782,-52.644,447.109,174.768,16.850,152.636
C07030=1089.777,-52.893,447.120,174.767,16.849,152.636
C07031=1089.770,-53.143,447.132,174.765,16.848,152.636
C07032=1089.764,-53.392,447.142,174.764,16.846,152.636
C07033=1089.758,-53.642,447.155,174.762,16.845,152.636
C07034=1089.753,-53.891,447.166,174.761,16.844,152.636
C07035=1089.746,-54.141,447.178,174.759,16.843,152.636
C07036=1089.740,-54.392,447.190,174.758,16.841,152.636
C07037=1089.734,-54.640,447.201,174.756,16.840,152.636
C07038=1089.728,-54.891,447.212,174.754,16.839,152.637
C07039=1089.722,-55.139,447.224,174.753,16.838,152.637
C07040=1089.716,-55.390,447.236,174.751,16.837,152.637
C07041=1089.710,-55.639,447.248,174.750,16.835,152.637
C07042=1089.704,-55.889,447.259,174.748,16.834,152.637
C07043=1089.698,-56.138,447.270,174.746,16.833,152.637
C07044=1089.692,-56.388,447.282,174.745,16.832,152.637
C07045=1089.686,-56.637,447.294,174.743,16.831,152.637
C07046=1089.680,-56.887,447.305,174.742,16.829,152.637
C07047=1089.674,-57.136,447.317,174.740,16.828,152.637
C07048=1089.668,-57.387,447.328,174.739,16.827,152.637
C07049=1089.663,-57.636,447.339,174.737,16.826,152.637
C07050=1089.656,-57.886,447.351,174.735,16.825,152.638
C07051=1089.650,-58.135,447.362,174.734,16.823,152.637
C07052=1089.644,-58.385,447.374,174.732,16.822,152.638
C07053=1089.639,-58.635,447.386,174.731,16.821,152.638
C07054=1089.632,-58.885,447.397,174.729,16.820,152.638
C07055=1089.626,-59.134,447.408,174.728,16.819,152.638
C07056=1089.620,-59.384,447.420,174.726,16.817,152.638
C07057=1089.614,-59.634,447.431,174.725,16.816,152.638
C07058=1089.608,-59.883,447.443,174.723,16.815,152.638
C07059=1089.602,-60.133,447.454,174.721,16.814,152.638
C07060=1089.596,-60.383,447.465,174.720,16.813,152.638
C07061=1089.590,-60.632,447.477,174.718,16.811,152.638
C07062=1089.584,-60.882,447.488,174.717,16.810,152.638
C07063=1089.579,-61.132,447.500,174.715,16.809,152.638
C07064=1089.573,-61.381,447.511,174.713,16.808,152.639
C07065=1089.566,-61.631,447.522,174.712,16.806,152.639
C07066=1089.561,-61.880,447.533,174.710,16.805,152.639
C07067=1089.554,-62.130,447.545,174.709,16.804,152.639
C07068=1089.548,-62.380,447.556,174.707,16.803,152.639
C07069=1089.543,-62.630,447.568,174.706,16.802,152.639
C07070=1089.537,-62.880,447.579,174.704,16.800,152.639
C07071=1089.531,-63.128,447.590,174.702,16.799,152.639
C07072=1089.524,-63.379,447.602,174.701,16.798,152.639
C07073=1089.519,-63.628,447.613,174.699,16.797,152.639
C07074=1089.512,-63.878,447.624,174.698,16.795,152.639
C07075=1089.507,-64.127,447.636,174.696,16.794,152.639
C07076=1089.501,-64.377,447.647,174.694,16.793,152.640
C07077=1089.495,-64.649,447.659,174.693,16.792,152.640
C07078=1089.489,-64.921,447.671,174.691,16.791,152.640
C07079=1089.482,-65.193,447.683,174.690,16.789,152.640
C07080=1089.475,-65.465,447.695,174.687,16.788,152.640
C07081=1089.469,-65.715,447.707,174.686,16.787,152.640
C07082=1089.463,-65.964,447.719,174.685,16.786,152.640
C07083=1089.458,-66.214,447.730,174.683,16.785,152.640
C07084=1089.451,-66.464,447.741,174.682,16.783,152.640
C07085=1089.446,-66.714,447.752,174.680,16.782,152.640
C07086=1089.440,-66.963,447.763,174.679,16.781,152.640
C07087=1089.434,-67.213,447.774,174.677,16.780,152.640
C07088=1089.427,-67.462,447.785,174.675,16.779,152.641
C07089=1089.422,-67.712,447.796,174.674,16.778,152.641
C07090=1089.415,-67.962,447.808,174.672,16.777,152.641
C07091=1089.410,-68.212,447.819,174.671,16.775,152.641
C07092=1089.405,-68.461,447.830,174.669,16.774,152.641
C07093=1089.398,-68.711,447.841,174.668,16.773,152.641
C07094=1089.393,-68.961,447.852,174.666,16.772,152.641
C07095=1089.387,-69.210,447.863,174.664,16.771,152.641
C07096=1089.380,-69.461,447.874,174.663,16.769,152.641
C07097=1089.375,-69.710,447.885,174.661,16.768,152.641
C07098=1089.369,-69.959,447.897,174.660,16.767,152.641
C07099=1089.362,-70.209,447.908,174.658,16.766,152.641
C07100=1089.357,-70.459,447.919,174.657,16.765,152.642
C07101=1089.351,-70.708,447.930,174.655,16.763,152.642
C07102=1089.345,-70.958,447.941,174.653,16.762,152.642
C07103=1089.339,-71.208,447.952,174.652,16.761,152.642
C07104=1089.334,-71.458,447.963,174.650,16.760,152.642
C07105=1089.328,-71.707,447.974,174.649,16.758,152.642
C07106=1089.322,-71.957,447.985,174.647,16.757,152.642
C07107=1089.316,-72.207,447.996,174.646,16.757,152.642
C07108=1089.310,-72.456,448.007,174.645,16.756,152.642
C07109=1089.304,-72.706,448.018,174.643,16.755,152.642
C07110=1089.298,-72.956,448.029,174.641,16.753,152.642
C07111=1089.292,-73.205,448.040,174.640,16.752,152.643
C07112=1089.287,-73.455,448.051,174.638,16.751,152.643
C07113=1089.281,-73.704,448.062,174.636,16.750,152.643
C07114=1089.275,-73.955,448.073,174.635,16.749,152.643
C07115=1089.269,-74.204,448.084,174.633,16.747,152.643
C07116=1089.263,-74.454,448.095,174.632,16.746,152.643
C07117=1089.257,-74.703,448.106,174.630,16.745,152.643
C07118=1089.251,-74.953,448.117,174.629,16.744,152.643
C07119=1089.245,-75.202,448.127,174.627,16.743,152.643
C07120=1089.239,-75.452,448.138,174.625,16.742,152.643
C07121=1089.233,-75.703,448.149,174.625,16.741,152.643
C07122=1089.227,-75.952,448.160,174.623,16.740,152.643
C07123=1089.221,-76.202,448.170,174.621,16.739,152.644
C07124=1089.216,-76.451,448.181,174.620,16.738,152.644
C07125=1089.209,-76.701,448.193,174.618,16.737,152.644
C07126=1089.203,-76.951,448.203,174.616,16.736,152.644
C07127=1089.197,-77.200,448.214,174.615,16.735,152.644
C07128=1089.191,-77.450,448.225,174.613,16.734,152.644
C07129=1089.185,-77.700,448.236,174.611,16.732,152.644
C07130=1089.179,-77.949,448.247,174.610,16.731,152.644
C07131=1089.174,-78.199,448.257,174.608,16.730,152.644
C07132=1089.167,-78.449,448.268,174.607,16.729,152.645
C07133=1089.161,-78.699,448.278,174.606,16.729,152.645
C07134=1089.155,-78.948,448.289,174.604,16.727,152.645
C07135=1089.149,-79.198,448.300,174.603,16.726,152.645
C07136=1089.144,-79.447,448.311,174.601,16.725,152.645
C07137=1089.137,-79.697,448.322,174.599,16.724,152.645
C07138=1089.131,-79.947,448.332,174.598,16.723,152.645
C07139=1089.125,-80.197,448.343,174.596,16.722,152.645
C07140=1089.120,-80.446,448.354,174.594,16.721,152.646
C07141=1089.112,-80.721,448.365,174.592,16.720,152.646
C07142=1089.106,-80.994,448.377,174.591,16.719,152.646
C07143=1089.099,-81.269,448.388,174.589,16.718,152.646
C07144=1089.092,-81.543,448.401,174.588,16.717,152.646
C07145=1089.086,-81.792,448.410,174.586,16.716,152.646
C07146=1089.080,-82.043,448.421,174.584,16.715,152.646
C07147=1089.074,-82.292,448.432,174.583,16.713,152.646
C07148=1089.068,-82.541,448.443,174.581,16.712,152.646
C07149=1089.062,-82.791,448.453,174.580,16.712,152.647
C07150=1089.056,-83.042,448.464,174.578,16.711,152.647
C07151=1089.049,-83.291,448.474,174.577,16.710,152.647
C07152=1089.044,-83.540,448.485,174.575,16.709,152.647
C07153=1089.038,-83.790,448.495,174.573,16.708,152.647
C07154=1089.031,-84.040,448.506,174.572,16.707,152.647
C07155=1089.025,-84.290,448.517,174.570,16.706,152.647
C07156=1089.019,-84.539,448.527,174.569,16.705,152.647
C07157=1089.014,-84.789,448.537,174.567,16.705,152.648
C07158=1089.008,-85.038,448.548,174.566,16.703,152.648
C07159=1089.001,-85.288,448.559,174.564,16.702,152.648
C07160=1088.995,-85.538,448.569,174.563,16.701,152.648
C07161=1088.989,-85.788,448.579,174.561,16.700,152.648
C07162=1088.983,-86.037,448.590,174.559,16.699,152.648
C07163=1088.978,-86.287,448.600,174.558,16.698,152.648
C07164=1088.971,-86.537,448.611,174.557,16.698,152.649
C07165=1088.965,-86.787,448.622,174.555,16.697,152.649
C07166=1088.959,-87.036,448.631,174.553,16.696,152.649
C07167=1088.953,-87.286,448.642,174.552,16.694,152.649
C07168=1088.946,-87.535,448.653,174.550,16.693,152.649
C07169=1088.940,-87.786,448.663,174.548,16.692,152.649
C07170=1088.935,-88.035,448.674,174.547,16.691,152.649
C07171=1088.928,-88.285,448.684,174.546,16.691,152.649
C07172=1088.923,-88.535,448.694,174.544,16.690,152.649
C07173=1088.916,-88.784,448.705,174.542,16.689,152.650
C07174=1088.911,-89.034,448.715,174.541,16.688,152.650
C07175=1088.904,-89.283,448.725,174.539,16.687,152.650
C07176=1088.898,-89.533,448.736,174.537,16.686,152.650
C07177=1088.893,-89.783,448.747,174.536,16.685,152.650
C07178=1088.886,-90.033,448.757,174.535,16.684,152.650
C07179=1088.881,-90.283,448.767,174.533,16.683,152.650
C07180=1088.874,-90.532,448.777,174.532,16.682,152.650
C07181=1088.869,-90.782,448.787,174.530,16.681,152.651
C07182=1088.862,-91.031,448.798,174.528,16.680,152.651
C07183=1088.856,-91.281,448.809,174.526,16.679,152.651
C07184=1088.850,-91.531,448.818,174.526,16.679,152.651
C07185=1088.844,-91.781,448.829,174.524,16.678,152.651
C07186=1088.838,-92.030,448.839,174.522,16.677,152.651
C07187=1088.832,-92.280,448.850,174.520,16.676,152.652
C07188=1088.826,-92.530,448.859,174.519,16.675,152.652
C07189=1088.820,-92.779,448.870,174.518,16.674,152.652
C07190=1088.814,-93.029,448.880,174.516,16.673,152.652
C07191=1088.808,-93.278,448.891,174.515,16.672,152.652
C07192=1088.803,-93.529,448.901,174.513,16.671,152.652
C07193=1088.796,-93.778,448.911,174.511,16.670,152.652
C07194=1088.790,-94.029,448.922,174.510,16.669,152.652
C07195=1088.784,-94.278,448.932,174.509,16.669,152.652
C07196=1088.778,-94.528,448.942,174.507,16.668,152.653
C07197=1088.772,-94.778,448.952,174.505,16.667,152.653
C07198=1088.767,-95.027,448.963,174.504,16.666,152.653
C07199=1088.760,-95.277,448.972,174.502,16.665,152.653
C07200=1088.754,-95.526,448.982,174.500,16.664,152.653
C07201=1088.748,-95.776,448.993,174.499,16.664,152.653
C07202=1088.742,-96.025,449.003,174.498,16.663,152.653
C07203=1088.737,-96.276,449.013,174.496,16.661,152.654
C07204=1088.730,-96.525,449.023,174.494,16.661,152.654
C07205=1088.724,-96.802,449.034,174.492,16.660,152.654
C07206=1088.717,-97.078,449.046,174.491,16.659,152.654
C07207=1088.711,-97.354,449.057,174.489,16.657,152.654
C07208=1088.704,-97.631,449.068,174.487,16.657,152.654
C07209=1088.698,-97.881,449.078,174.486,16.656,152.655
C07210=1088.692,-98.130,449.088,174.485,16.655,152.655
C07211=1088.686,-98.380,449.098,174.483,16.655,152.655
C07212=1088.680,-98.630,449.108,174.481,16.653,152.655
C07213=1088.673,-98.879,449.118,174.480,16.652,152.655
C07214=1088.668,-99.130,449.129,174.479,16.652,152.655
C07215=1088.662,-99.379,449.138,174.477,16.651,152.655
C07216=1088.655,-99.629,449.148,174.475,16.650,152.656
C07217=1088.649,-99.878,449.158,174.473,16.650,152.656
C07218=1088.643,-100.128,449.168,174.472,16.648,152.656
C07219=1088.637,-100.378,449.178,174.471,16.648,152.656
C07220=1088.631,-100.627,449.188,174.469,16.647,152.656
C07221=1088.625,-100.878,449.198,174.467,16.646,152.656
C07222=1088.619,-101.127,449.208,174.465,16.646,152.657
C07223=1088.613,-101.377,449.218,174.464,16.644,152.657
C07224=1088.607,-101.626,449.228,174.463,16.644,152.657
C07225=1088.601,-101.876,449.238,174.461,16.643,152.657
C07226=1088.595,-102.126,449.248,174.459,16.642,152.657
C07227=1088.588,-102.375,449.258,174.458,16.642,152.657
C07228=1088.583,-102.626,449.268,174.457,16.641,152.658
C07229=1088.577,-102.875,449.278,174.455,16.640,152.658
C07230=1088.570,-103.125,449.288,174.453,16.639,152.658
C07231=1088.564,-103.374,449.297,174.452,16.638,152.658
C07232=1088.559,-103.624,449.307,174.450,16.638,152.658
C07233=1088.552,-103.874,449.318,174.449,16.637,152.658
C07234=1088.546,-104.123,449.327,174.447,16.636,152.658
C07235=1088.540,-104.373,449.337,174.445,16.635,152.659
C07236=1088.534,-104.623,449.346,174.444,16.635,152.659
C07237=1088.528,-104.872,449.357,174.443,16.634,152.659
C07238=1088.522,-105.122,449.367,174.441,16.633,152.659
C07239=1088.516,-105.372,449.376,174.439,16.632,152.659
C07240=1088.510,-105.622,449.386,174.438,16.632,152.659
C07241=1088.504,-105.872,449.396,174.437,16.631,152.660
C07242=1088.498,-106.121,449.406,174.435,16.630,152.660
C07243=1088.491,-106.371,449.416,174.433,16.629,152.660
C07244=1088.485,-106.621,449.425,174.432,16.629,152.660
C07245=1088.479,-106.871,449.435,174.430,16.628,152.660
C07246=1088.474,-107.121,449.445,174.428,16.627,152.661
C07247=1088.468,-107.370,449.455,174.427,16.626,152.661
C07248=1088.461,-107.620,449.465,174.426,16.626,152.661
C07249=1088.455,-107.869,449.475,174.424,16.625,152.661
C07250=1088.449,-108.119,449.484,174.422,16.625,152.661
C07251=1088.443,-108.369,449.494,174.420,16.623,152.661
C07252=1088.436,-108.619,449.503,174.419,16.623,152.662
C07253=1088.430,-108.869,449.513,174.418,16.622,152.662
C07254=1088.424,-109.118,449.522,174.416,16.622,152.662
C07255=1088.419,-109.369,449.533,174.414,16.621,152.662
C07256=1088.412,-109.618,449.543,174.413,16.621,152.662
C07257=1088.406,-109.868,449.552,174.411,16.619,152.662
C07258=1088.400,-110.117,449.562,174.410,16.619,152.663
C07259=1088.394,-110.367,449.572,174.409,16.618,152.663
C07260=1088.387,-110.617,449.581,174.407,16.618,152.663
C07261=1088.381,-110.867,449.591,174.405,16.617,152.663
C07262=1088.375,-111.117,449.600,174.403,16.616,152.663
C07263=1088.370,-111.366,449.610,174.402,16.615,152.663
C07264=1088.363,-111.615,449.619,174.401,16.615,152.664
C07265=1088.357,-111.865,449.629,174.399,16.614,152.664
C07266=1088.351,-112.115,449.638,174.397,16.613,152.664
C07267=1088.345,-112.365,449.648,174.396,16.613,152.664
C07268=1088.339,-112.615,449.657,174.394,16.612,152.664
C07269=1088.332,-112.885,449.668,174.392,16.611,152.665
C07270=1088.325,-113.156,449.679,174.390,16.611,152.665
C07271=1088.319,-113.427,449.689,174.390,16.610,152.665
C07272=1088.312,-113.696,449.699,174.388,16.610,152.665
C07273=1088.306,-113.946,449.709,174.386,16.608,152.665
C07274=1088.300,-114.196,449.718,174.384,16.608,152.666
C07275=1088.294,-114.446,449.728,174.383,16.608,152.666
C07276=1088.288,-114.696,449.737,174.381,16.607,152.666
C07277=1088.282,-114.945,449.747,174.380,16.606,152.666
